Yaskawa INFORM job: aprem3TRJ3.JBI

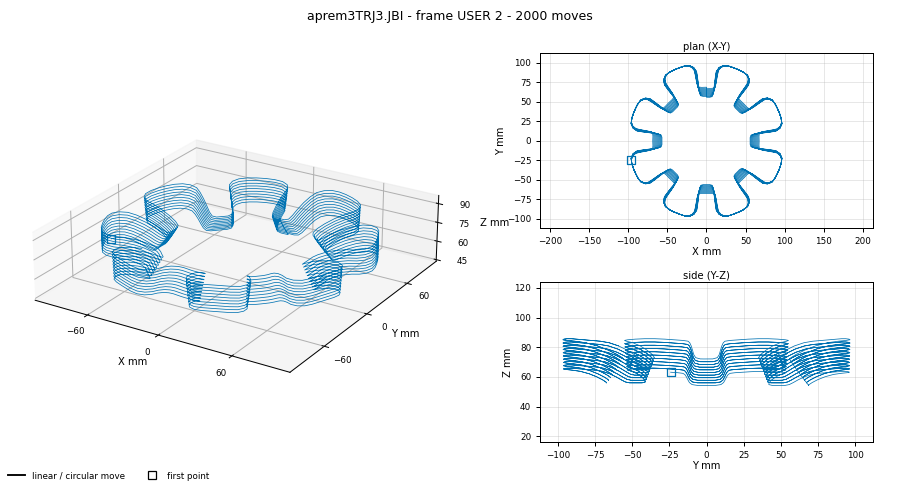
[picture p0: tool path of aprem3TRJ3.JBI in frame USER 2, 2000 of 2000 moves have a stored position in this frame; points joined in program order, loops and branches not executed]
/JOB
//NAME aprem3TRJ3
///FOLDERNAME DEMO
//POS
///NPOS 2000,0,2000,0,0,0
///USER 2
///TOOL 7
///POSTYPE USER
///RECTAN
///RCONF 1,0,0,0,0,0,0,0,0,0,0,0,0,0,0,0,0,0,0,0,0,0,0,0
C00000=-96.154,-24.159,63.210,179.7472,-2.4641,-10695.8962
C00001=-94.423,-19.246,62.877,177.2942,-4.1530,-10698.4794
C00002=-90.636,-15.942,62.469,172.7045,-3.4321,-10700.0243
C00003=-85.405,-14.621,61.698,172.2425,-1.7901,-10700.2854
C00004=-79.780,-13.569,60.151,174.0266,-1.3203,-10700.3475
C00005=-74.809,-12.586,58.158,176.9961,-0.7607,-10700.4499
C00006=-71.127,-11.507,56.252,-176.5790,1.2623,-10700.8103
C00007=-69.044,-9.699,54.888,-163.7838,26.3525,-10702.0037
C00008=-68.619,-6.200,54.350,-178.9508,38.3093,-10704.8371
C00009=-68.781,-2.945,54.326,177.7405,38.7530,-10707.5483
C00010=-68.843,0.000,54.342,179.9996,38.7765,-10710.0000
C00011=-68.781,2.945,54.326,-177.7401,38.7530,-10712.4517
C00012=-68.619,6.200,54.350,178.9482,38.3089,-10715.1629
C00013=-69.044,9.699,54.888,163.7840,26.3528,-10717.9963
C00014=-71.127,11.507,56.252,176.5790,1.2623,-10719.1897
C00015=-74.809,12.586,58.158,-176.9961,-0.7607,-10719.5501
C00016=-79.780,13.569,60.151,-174.0266,-1.3203,-10719.6525
C00017=-85.405,14.621,61.698,-172.2425,-1.7901,-10719.7146
C00018=-90.636,15.942,62.469,-172.7045,-3.4321,-10719.9757
C00019=-94.423,19.246,62.877,-177.2942,-4.1530,-10721.5206
C00020=-96.154,24.159,63.210,-179.7472,-2.4641,-10724.1038
C00021=-95.429,29.718,63.547,179.9546,-0.1514,-10727.2974
C00022=-93.512,35.416,63.770,179.9933,-0.0179,-10730.7433
C00023=-91.166,41.080,63.770,179.9921,-0.0174,-10734.2566
C00024=-88.493,46.465,63.547,179.9251,-0.1391,-10737.7026
C00025=-85.074,50.908,63.210,178.0786,-1.5643,-10740.8962
C00026=-80.376,53.158,62.877,175.1551,-1.0270,-10743.4793
C00027=-75.362,52.817,62.469,172.4279,2.7549,-10745.0245
C00028=-70.729,50.052,61.698,173.2462,4.2451,-10745.2855
C00029=-66.007,46.818,60.151,174.8410,3.3018,-10745.3476
C00030=-61.798,43.998,58.158,177.3380,1.5877,-10745.4495
C00031=-58.431,42.158,56.252,-176.6891,-1.5289,-10745.8105
C00032=-55.679,41.963,54.888,-150.9290,8.2296,-10747.0038
C00033=-52.905,44.137,54.350,-150.2488,28.6202,-10749.8372
C00034=-50.718,46.553,54.326,-151.6454,30.7727,-10752.5482
C00035=-48.679,48.679,54.342,-150.4014,29.5989,-10755.0000
C00036=-46.553,50.718,54.326,-149.2271,28.3544,-10757.4518
C00037=-44.137,52.905,54.350,-151.3816,29.7523,-10760.1628
C00038=-41.963,55.680,54.888,-171.7700,29.0711,-10762.9966
C00039=-42.158,58.431,56.252,178.4711,3.3109,-10764.1895
C00040=-43.998,61.798,58.158,-178.4123,-2.6620,-10764.5505
C00041=-46.818,66.007,60.151,-176.6982,-5.1590,-10764.6524
C00042=-50.052,70.729,61.698,-175.7549,-6.7538,-10764.7145
C00043=-52.817,75.362,62.469,-177.2451,-7.5721,-10764.9755
C00044=-53.158,80.376,62.877,178.9730,-4.8449,-10766.5207
C00045=-50.908,85.074,63.210,178.4357,-1.9214,-10769.1038
C00046=-46.465,88.493,63.547,179.8609,-0.0749,-10772.2974
C00047=-41.080,91.166,63.770,179.9826,-0.0079,-10775.7434
C00048=-35.416,93.512,63.770,179.9821,-0.0067,-10779.2567
C00049=-29.718,95.429,63.547,179.8486,-0.0454,-10782.7026
C00050=-24.159,96.154,63.210,177.5359,0.2528,-10785.8962
C00051=-19.246,94.423,62.877,175.8470,2.7058,-10788.4794
C00052=-15.942,90.636,62.469,176.5679,7.2955,-10790.0243
C00053=-14.621,85.405,61.698,178.2099,7.7575,-10790.2854
C00054=-13.569,79.780,60.151,178.6797,5.9734,-10790.3475
C00055=-12.586,74.809,58.158,179.2393,3.0039,-10790.4499
C00056=-11.507,71.127,56.252,-178.7377,-3.4210,-10790.8103
C00057=-9.699,69.044,54.888,-153.6472,-16.2160,-10792.0037
C00058=-6.200,68.619,54.350,-141.6911,-1.0518,-10794.8371
C00059=-2.945,68.781,54.326,-141.2470,2.2599,-10797.5483
C00060=0.000,68.843,54.342,-141.2235,-0.0004,-10800.0000
C00061=0.000,67.469,56.061,-141.5412,-0.0004,-10800.0000
C00062=2.820,67.413,56.044,-141.5636,-2.1988,-10802.3954
C00063=5.989,67.263,56.069,-142.0566,1.4090,-10805.0881
C00064=9.441,67.734,56.637,-154.9636,16.3668,-10807.9350
C00065=11.191,69.937,58.076,-179.1454,2.5065,-10809.0911
C00066=12.227,73.809,60.085,179.1943,-3.3815,-10809.4060
C00067=13.183,79.025,62.181,178.7261,-6.0865,-10809.4709
C00068=14.211,84.918,63.804,178.3204,-7.7435,-10809.5004
C00069=15.500,90.396,64.610,176.7328,-7.3164,-10809.7298
C00070=18.832,94.373,65.037,175.8897,-2.7823,-10811.2851
C00071=23.832,96.213,65.385,177.5484,-0.2740,-10813.9122
C00072=29.513,95.497,65.736,179.8479,0.0454,-10817.1736
C00073=35.347,93.539,65.969,179.9821,0.0067,-10820.7008
C00074=41.148,91.136,65.969,179.9826,0.0079,-10824.2992
C00075=46.658,88.395,65.736,179.8603,0.0754,-10827.8267
C00076=51.181,84.885,65.385,178.4595,1.9277,-10831.0877
C00077=53.416,80.048,65.037,179.0575,4.8686,-10833.7152
C00078=52.959,74.880,64.610,-177.1134,7.4719,-10835.2699
C00079=49.997,70.095,63.804,-175.6871,6.6669,-10835.4993
C00080=46.557,65.200,62.181,-176.5849,5.2066,-10835.5293
C00081=43.545,60.837,60.085,-178.1765,2.9610,-10835.5938
C00082=41.540,57.367,58.076,178.8310,-2.3765,-10835.9087
C00083=41.220,54.571,56.637,-173.0100,-28.2777,-10837.0654
C00084=43.327,51.796,56.069,-151.9006,-29.6278,-10839.9123
C00085=45.674,49.662,56.044,-149.5306,-28.1035,-10842.6047
C00086=47.708,47.708,56.061,-150.6800,-29.3196,-10845.0000
C00087=49.662,45.674,56.044,-151.8968,-30.4697,-10847.3953
C00088=51.797,43.327,56.069,-150.3712,-28.0975,-10850.0883
C00089=54.571,41.220,56.637,-151.7222,-6.9903,-10852.9346
C00090=57.367,41.540,58.076,-177.6235,1.1690,-10854.0913
C00091=60.837,43.545,60.085,177.0390,-1.8235,-10854.4062
C00092=65.200,46.557,62.181,174.7934,-3.4151,-10854.4707
C00093=70.095,49.997,63.804,173.3331,-4.3129,-10854.5007
C00094=74.880,52.959,64.610,172.5281,-2.8866,-10854.7301
C00095=80.048,53.416,65.037,175.1314,0.9425,-10856.2848
C00096=84.885,51.181,65.385,178.0723,1.5405,-10858.9123
C00097=88.395,46.658,65.736,179.9246,0.1397,-10862.1733
C00098=91.136,41.148,65.969,179.9921,0.0174,-10865.7008
C00099=93.539,35.347,65.969,179.9933,0.0179,-10869.2992
C00100=95.497,29.513,65.736,179.9546,0.1521,-10872.8264
C00101=96.213,23.832,65.385,-179.7260,2.4516,-10876.0878
C00102=94.373,18.832,65.037,-177.2177,4.1103,-10878.7149
C00103=90.396,15.500,64.610,-172.6836,3.2672,-10880.2702
C00104=84.918,14.211,63.804,-172.2565,1.6796,-10880.4996
C00105=79.025,13.183,62.181,-173.9135,1.2739,-10880.5291
C00106=73.809,12.227,60.085,-176.6185,0.8057,-10880.5940
C00107=69.937,11.191,58.076,177.4935,-0.8546,-10880.9089
C00108=67.734,9.441,56.637,163.6332,-25.0364,-10882.0650
C00109=67.263,5.989,56.069,178.5910,-37.9434,-10884.9119
C00110=67.413,2.820,56.044,-177.8012,-38.4364,-10887.6046
C00111=67.469,0.000,56.061,-179.9996,-38.4588,-10890.0000
C00112=67.413,-2.820,56.044,177.8008,-38.4364,-10892.3954
C00113=67.263,-5.989,56.069,-178.5883,-37.9429,-10895.0881
C00114=67.734,-9.441,56.637,-163.6333,-25.0366,-10897.9350
C00115=69.937,-11.191,58.076,-177.4935,-0.8546,-10899.0911
C00116=73.809,-12.227,60.085,176.6185,0.8057,-10899.4060
C00117=79.025,-13.183,62.181,173.9135,1.2739,-10899.4709
C00118=84.918,-14.211,63.804,172.2565,1.6796,-10899.5004
C00119=90.396,-15.500,64.610,172.6836,3.2672,-10899.7298
C00120=94.373,-18.832,65.037,177.2177,4.1103,-10901.2851
C00121=96.213,-23.832,65.385,179.7260,2.4516,-10903.9122
C00122=95.497,-29.513,65.736,-179.9546,0.1521,-10907.1736
C00123=93.539,-35.347,65.969,-179.9933,0.0179,-10910.7008
C00124=91.136,-41.148,65.969,-179.9921,0.0174,-10914.2992
C00125=88.395,-46.658,65.736,-179.9246,0.1397,-10917.8267
C00126=84.885,-51.181,65.385,-178.0723,1.5405,-10921.0877
C00127=80.048,-53.416,65.037,-175.1314,0.9425,-10923.7152
C00128=74.880,-52.959,64.610,-172.5281,-2.8866,-10925.2699
C00129=70.095,-49.997,63.804,-173.3331,-4.3129,-10925.4993
C00130=65.200,-46.557,62.181,-174.7934,-3.4151,-10925.5293
C00131=60.837,-43.545,60.085,-177.0390,-1.8235,-10925.5938
C00132=57.367,-41.540,58.076,177.6235,1.1690,-10925.9087
C00133=54.571,-41.220,56.637,151.7223,-6.9900,-10927.0654
C00134=51.796,-43.327,56.069,150.3722,-28.0994,-10929.9123
C00135=49.662,-45.674,56.044,151.8965,-30.4694,-10932.6047
C00136=47.708,-47.708,56.061,150.6804,-29.3200,-10935.0000
C00137=45.674,-49.662,56.044,149.5303,-28.1032,-10937.3953
C00138=43.327,-51.797,56.069,151.9025,-29.6288,-10940.0883
C00139=41.220,-54.571,56.637,173.0097,-28.2778,-10942.9346
C00140=41.540,-57.367,58.076,-178.8310,-2.3765,-10944.0913
C00141=43.545,-60.837,60.085,178.1765,2.9610,-10944.4062
C00142=46.557,-65.200,62.181,176.5849,5.2066,-10944.4707
C00143=49.997,-70.095,63.804,175.6871,6.6669,-10944.5007
C00144=52.959,-74.880,64.610,177.1134,7.4719,-10944.7301
C00145=53.416,-80.048,65.037,-179.0575,4.8686,-10946.2848
C00146=51.181,-84.885,65.385,-178.4595,1.9277,-10948.9123
C00147=46.658,-88.395,65.736,-179.8603,0.0754,-10952.1733
C00148=41.148,-91.136,65.969,-179.9826,0.0079,-10955.7008
C00149=35.347,-93.539,65.969,-179.9821,0.0067,-10959.2992
C00150=29.513,-95.497,65.736,-179.8479,0.0454,-10962.8264
C00151=23.832,-96.213,65.385,-177.5484,-0.2740,-10966.0878
C00152=18.832,-94.373,65.037,-175.8897,-2.7823,-10968.7149
C00153=15.500,-90.396,64.610,-176.7328,-7.3164,-10970.2702
C00154=14.211,-84.918,63.804,-178.3204,-7.7435,-10970.4996
C00155=13.183,-79.025,62.181,-178.7261,-6.0865,-10970.5291
C00156=12.227,-73.809,60.085,-179.1943,-3.3815,-10970.5940
C00157=11.191,-69.937,58.076,179.1454,2.5065,-10970.9089
C00158=9.441,-67.734,56.637,154.9636,16.3668,-10972.0650
C00159=5.989,-67.263,56.069,142.0566,1.4090,-10974.9119
C00160=2.820,-67.413,56.044,141.5636,-2.1988,-10977.6046
C00161=0.000,-67.469,56.061,141.5412,-0.0004,-10980.0000
C00162=0.000,-67.469,56.061,141.5412,-0.0004,-10980.0000
C00163=-2.820,-67.413,56.044,141.5636,2.1992,-10982.3954
C00164=-5.989,-67.263,56.069,142.0571,-1.4117,-10985.0881
C00165=-9.441,-67.734,56.637,154.9634,-16.3667,-10987.9350
C00166=-11.191,-69.937,58.076,179.1454,-2.5065,-10989.0911
C00167=-12.227,-73.809,60.085,-179.1943,3.3815,-10989.4060
C00168=-13.183,-79.025,62.181,-178.7261,6.0865,-10989.4709
C00169=-14.211,-84.918,63.804,-178.3204,7.7435,-10989.5004
C00170=-15.500,-90.396,64.610,-176.7328,7.3164,-10989.7298
C00171=-18.832,-94.373,65.037,-175.8897,2.7823,-10991.2851
C00172=-23.832,-96.213,65.385,-177.5484,0.2740,-10993.9122
C00173=-29.513,-95.497,65.736,-179.8479,-0.0454,-10997.1736
C00174=-35.347,-93.539,65.969,-179.9821,-0.0067,-11000.7008
C00175=-41.148,-91.136,65.969,-179.9826,-0.0079,-11004.2992
C00176=-46.658,-88.395,65.736,-179.8603,-0.0754,-11007.8267
C00177=-51.181,-84.885,65.385,-178.4595,-1.9277,-11011.0877
C00178=-53.416,-80.048,65.037,-179.0575,-4.8686,-11013.7152
C00179=-52.959,-74.880,64.610,177.1134,-7.4719,-11015.2699
C00180=-49.997,-70.095,63.804,175.6871,-6.6669,-11015.4993
C00181=-46.557,-65.200,62.181,176.5849,-5.2066,-11015.5293
C00182=-43.545,-60.837,60.085,178.1765,-2.9610,-11015.5938
C00183=-41.540,-57.367,58.076,-178.8310,2.3765,-11015.9087
C00184=-41.220,-54.571,56.637,173.0100,28.2777,-11017.0654
C00185=-43.327,-51.796,56.069,151.9006,29.6278,-11019.9123
C00186=-45.674,-49.662,56.044,149.5306,28.1035,-11022.6047
C00187=-47.708,-47.708,56.061,150.6800,29.3196,-11025.0000
C00188=-49.662,-45.674,56.044,151.8968,30.4697,-11027.3953
C00189=-51.797,-43.327,56.069,150.3712,28.0975,-11030.0883
C00190=-54.571,-41.220,56.637,151.7222,6.9903,-11032.9346
C00191=-57.367,-41.540,58.076,177.6235,-1.1690,-11034.0913
C00192=-60.837,-43.545,60.085,-177.0390,1.8235,-11034.4062
C00193=-65.200,-46.557,62.181,-174.7934,3.4151,-11034.4707
C00194=-70.095,-49.997,63.804,-173.3331,4.3129,-11034.5007
C00195=-74.880,-52.959,64.610,-172.5281,2.8866,-11034.7301
C00196=-80.048,-53.416,65.037,-175.1314,-0.9425,-11036.2848
C00197=-84.885,-51.181,65.385,-178.0723,-1.5405,-11038.9123
C00198=-88.395,-46.658,65.736,-179.9246,-0.1397,-11042.1733
C00199=-91.136,-41.148,65.969,-179.9921,-0.0174,-11045.7008
C00200=-93.539,-35.347,65.969,-179.9933,-0.0179,-11049.2992
C00201=-95.497,-29.513,65.736,-179.9546,-0.1521,-11052.8264
C00202=-96.213,-23.832,65.385,179.7260,-2.4516,-11056.0878
C00203=-94.373,-18.832,65.037,177.2177,-4.1103,-11058.7149
C00204=-90.396,-15.500,64.610,172.6836,-3.2672,-11060.2702
C00205=-84.918,-14.211,63.804,172.2565,-1.6796,-11060.4996
C00206=-79.025,-13.183,62.181,173.9135,-1.2739,-11060.5291
C00207=-73.809,-12.227,60.085,176.6185,-0.8057,-11060.5940
C00208=-69.937,-11.191,58.076,-177.4935,0.8546,-11060.9089
C00209=-67.734,-9.441,56.637,-163.6332,25.0364,-11062.0650
C00210=-67.263,-5.989,56.069,-178.5910,37.9434,-11064.9119
C00211=-67.413,-2.820,56.044,177.8012,38.4364,-11067.6046
C00212=-67.469,0.000,56.061,179.9996,38.4588,-11070.0000
C00213=-67.413,2.820,56.044,-177.8008,38.4364,-11072.3954
C00214=-67.263,5.989,56.069,178.5883,37.9429,-11075.0881
C00215=-67.734,9.441,56.637,163.6333,25.0366,-11077.9350
C00216=-69.937,11.191,58.076,177.4935,0.8546,-11079.0911
C00217=-73.809,12.227,60.085,-176.6185,-0.8057,-11079.4060
C00218=-79.025,13.183,62.181,-173.9135,-1.2739,-11079.4709
C00219=-84.918,14.211,63.804,-172.2565,-1.6796,-11079.5004
C00220=-90.396,15.500,64.610,-172.6836,-3.2672,-11079.7298
C00221=-94.373,18.832,65.037,-177.2177,-4.1103,-11081.2851
C00222=-96.213,23.832,65.385,-179.7260,-2.4516,-11083.9122
C00223=-95.497,29.513,65.736,179.9546,-0.1521,-11087.1736
C00224=-93.539,35.347,65.969,179.9933,-0.0179,-11090.7008
C00225=-91.136,41.148,65.969,179.9921,-0.0174,-11094.2992
C00226=-88.395,46.658,65.736,179.9246,-0.1397,-11097.8267
C00227=-84.885,51.181,65.385,178.0723,-1.5405,-11101.0877
C00228=-80.048,53.416,65.037,175.1314,-0.9425,-11103.7152
C00229=-74.880,52.959,64.610,172.5281,2.8866,-11105.2699
C00230=-70.095,49.997,63.804,173.3331,4.3129,-11105.4993
C00231=-65.200,46.557,62.181,174.7934,3.4151,-11105.5293
C00232=-60.837,43.545,60.085,177.0390,1.8235,-11105.5938
C00233=-57.367,41.540,58.076,-177.6235,-1.1690,-11105.9087
C00234=-54.571,41.220,56.637,-151.7223,6.9900,-11107.0654
C00235=-51.796,43.327,56.069,-150.3722,28.0994,-11109.9123
C00236=-49.662,45.674,56.044,-151.8965,30.4694,-11112.6047
C00237=-47.708,47.708,56.061,-150.6804,29.3200,-11115.0000
C00238=-45.674,49.662,56.044,-149.5303,28.1032,-11117.3953
C00239=-43.327,51.797,56.069,-151.9025,29.6288,-11120.0883
C00240=-41.220,54.571,56.637,-173.0097,28.2778,-11122.9346
C00241=-41.540,57.367,58.076,178.8310,2.3765,-11124.0913
C00242=-43.545,60.837,60.085,-178.1765,-2.9610,-11124.4062
C00243=-46.557,65.200,62.181,-176.5849,-5.2066,-11124.4707
C00244=-49.997,70.095,63.804,-175.6871,-6.6669,-11124.5007
C00245=-52.959,74.880,64.610,-177.1134,-7.4719,-11124.7301
C00246=-53.416,80.048,65.037,179.0575,-4.8686,-11126.2848
C00247=-51.181,84.885,65.385,178.4595,-1.9277,-11128.9123
C00248=-46.658,88.395,65.736,179.8603,-0.0754,-11132.1733
C00249=-41.148,91.136,65.969,179.9826,-0.0079,-11135.7008
C00250=-35.347,93.539,65.969,179.9821,-0.0067,-11139.2992
C00251=-29.513,95.497,65.736,179.8479,-0.0454,-11142.8264
C00252=-23.832,96.213,65.385,177.5484,0.2740,-11146.0878
C00253=-18.832,94.373,65.037,175.8897,2.7823,-11148.7149
C00254=-15.500,90.396,64.610,176.7328,7.3164,-11150.2702
C00255=-14.211,84.918,63.804,178.3204,7.7435,-11150.4996
C00256=-13.183,79.025,62.181,178.7261,6.0865,-11150.5291
C00257=-12.227,73.809,60.085,179.1943,3.3815,-11150.5940
C00258=-11.191,69.937,58.076,-179.1454,-2.5065,-11150.9089
C00259=-9.441,67.734,56.637,-154.9634,-16.3667,-11152.0650
C00260=-5.989,67.263,56.069,-142.0571,-1.4117,-11154.9119
C00261=-2.820,67.413,56.044,-141.5636,2.1992,-11157.6046
C00262=0.000,67.469,56.061,-141.5412,-0.0004,-11160.0000
C00263=0.000,66.107,57.788,-141.9405,-0.0005,-11160.0000
C00264=2.695,66.055,57.771,-141.9617,-2.1301,-11162.3363
C00265=5.779,65.917,57.797,-142.5088,1.7632,-11165.0104
C00266=9.185,66.436,58.394,-156.3340,16.3865,-11167.8714
C00267=10.880,68.762,59.909,-179.4729,1.6691,-11168.9912
C00268=11.874,72.826,62.021,179.1708,-3.6886,-11169.2604
C00269=12.805,78.288,64.219,178.7806,-6.1350,-11169.2892
C00270=13.814,84.445,65.915,178.4333,-7.6593,-11169.2905
C00271=15.073,90.163,66.756,176.9116,-7.2599,-11169.4907
C00272=18.432,94.325,67.200,175.9710,-2.8231,-11171.0568
C00273=23.517,96.271,67.561,177.5835,-0.2906,-11173.7273
C00274=29.315,95.562,67.927,179.8488,0.0450,-11177.0541
C00275=35.280,93.564,68.167,179.9823,0.0066,-11180.6599
C00276=41.213,91.107,68.167,179.9828,0.0078,-11184.3400
C00277=46.844,88.301,67.927,179.8613,0.0751,-11187.9461
C00278=51.445,84.703,67.561,178.4961,1.9145,-11191.2727
C00279=53.664,79.731,67.200,179.1443,4.8399,-11193.9430
C00280=53.097,74.413,66.756,-177.0274,7.3072,-11195.5096
C00281=49.944,69.479,65.915,-175.6680,6.5281,-11195.7099
C00282=46.303,64.413,64.219,-176.5119,5.2027,-11195.7103
C00283=43.100,59.892,62.021,-177.9754,3.1949,-11195.7399
C00284=40.929,56.315,59.909,179.1922,-1.5529,-11196.0092
C00285=40.483,53.472,58.394,-174.1779,-27.3765,-11197.1289
C00286=42.524,50.697,57.797,-152.4966,-29.4307,-11199.9895
C00287=44.802,48.614,57.771,-149.9071,-27.7853,-11202.6632
C00288=46.745,46.745,57.788,-151.0292,-28.9702,-11205.0000
C00289=48.613,44.802,57.771,-152.2149,-30.0932,-11207.3362
C00290=50.697,42.524,57.797,-150.5682,-27.5015,-11210.0105
C00291=53.472,40.483,58.395,-152.6235,-5.8223,-11212.8711
C00292=56.315,40.929,59.909,-178.4471,0.8078,-11213.9908
C00293=59.892,43.100,62.021,176.8051,-2.0246,-11214.2601
C00294=64.413,46.303,64.219,174.7973,-3.4881,-11214.2897
C00295=69.479,49.944,65.915,173.4719,-4.3320,-11214.2901
C00296=74.413,53.097,66.756,172.6928,-2.9726,-11214.4904
C00297=79.731,53.664,67.200,175.1601,0.8557,-11216.0570
C00298=84.703,51.445,67.561,178.0855,1.5039,-11218.7273
C00299=88.301,46.844,67.927,179.9249,0.1387,-11222.0539
C00300=91.107,41.213,68.167,179.9922,0.0172,-11225.6600
C00301=93.564,35.280,68.167,179.9934,0.0177,-11229.3401
C00302=95.562,29.315,67.927,179.9550,0.1512,-11232.9459
C00303=96.271,23.517,67.561,-179.7094,2.4165,-11236.2727
C00304=94.325,18.432,67.200,-177.1769,4.0290,-11238.9432
C00305=90.163,15.073,66.756,-172.7401,3.0884,-11240.5093
C00306=84.445,13.814,65.915,-172.3407,1.5667,-11240.7095
C00307=78.288,12.805,64.219,-173.8650,1.2194,-11240.7108
C00308=72.826,11.874,62.021,-176.3114,0.8292,-11240.7396
C00309=68.762,10.880,59.909,178.3309,-0.5271,-11241.0088
C00310=66.436,9.185,58.394,163.6135,-23.6660,-11242.1286
C00311=65.917,5.779,57.797,178.2368,-37.4912,-11244.9896
C00312=66.055,2.695,57.771,-177.8699,-38.0383,-11247.6637
C00313=66.107,0.000,57.788,-179.9995,-38.0595,-11250.0000
C00314=66.055,-2.695,57.771,177.8693,-38.0383,-11252.3363
C00315=65.917,-5.780,57.797,-178.2340,-37.4907,-11255.0112
C00316=66.436,-9.185,58.395,-163.6136,-23.6662,-11257.8714
C00317=68.762,-10.880,59.909,-178.3309,-0.5271,-11258.9912
C00318=72.826,-11.874,62.021,176.3114,0.8292,-11259.2604
C00319=78.288,-12.805,64.219,173.8650,1.2194,-11259.2892
C00320=84.445,-13.814,65.915,172.3407,1.5667,-11259.2905
C00321=90.163,-15.073,66.756,172.7401,3.0884,-11259.4907
C00322=94.325,-18.432,67.200,177.1769,4.0290,-11261.0568
C00323=96.271,-23.517,67.561,179.7094,2.4165,-11263.7273
C00324=95.562,-29.315,67.927,-179.9550,0.1512,-11267.0541
C00325=93.564,-35.280,68.167,-179.9934,0.0177,-11270.6599
C00326=91.107,-41.213,68.167,-179.9922,0.0172,-11274.3400
C00327=88.301,-46.844,67.927,-179.9249,0.1387,-11277.9461
C00328=84.703,-51.445,67.561,-178.0855,1.5039,-11281.2727
C00329=79.731,-53.664,67.200,-175.1601,0.8557,-11283.9430
C00330=74.413,-53.097,66.756,-172.6928,-2.9726,-11285.5096
C00331=69.479,-49.944,65.915,-173.4719,-4.3320,-11285.7099
C00332=64.413,-46.303,64.219,-174.7973,-3.4881,-11285.7103
C00333=59.892,-43.100,62.021,-176.8051,-2.0246,-11285.7399
C00334=56.315,-40.929,59.909,178.4471,0.8078,-11286.0092
C00335=53.472,-40.483,58.394,152.6235,-5.8221,-11287.1289
C00336=50.697,-42.524,57.797,150.5693,-27.5034,-11289.9895
C00337=48.614,-44.802,57.771,152.2147,-30.0929,-11292.6632
C00338=46.745,-46.745,57.788,151.0298,-28.9708,-11295.0000
C00339=44.802,-48.613,57.771,149.9068,-27.7851,-11297.3362
C00340=42.524,-50.697,57.797,152.4985,-29.4318,-11300.0105
C00341=40.483,-53.472,58.395,174.1777,-27.3765,-11302.8711
C00342=40.929,-56.315,59.909,-179.1922,-1.5529,-11303.9908
C00343=43.100,-59.892,62.021,177.9754,3.1949,-11304.2601
C00344=46.303,-64.413,64.219,176.5119,5.2027,-11304.2897
C00345=49.944,-69.479,65.915,175.6680,6.5281,-11304.2901
C00346=53.097,-74.413,66.756,177.0274,7.3072,-11304.4904
C00347=53.664,-79.731,67.200,-179.1443,4.8399,-11306.0570
C00348=51.445,-84.703,67.561,-178.4961,1.9145,-11308.7273
C00349=46.844,-88.301,67.927,-179.8613,0.0751,-11312.0539
C00350=41.213,-91.107,68.167,-179.9828,0.0078,-11315.6600
C00351=35.280,-93.564,68.167,-179.9823,0.0066,-11319.3401
C00352=29.315,-95.562,67.927,-179.8488,0.0450,-11322.9459
C00353=23.517,-96.271,67.561,-177.5835,-0.2906,-11326.2727
C00354=18.432,-94.325,67.200,-175.9710,-2.8231,-11328.9432
C00355=15.073,-90.163,66.756,-176.9116,-7.2599,-11330.5093
C00356=13.814,-84.445,65.915,-178.4333,-7.6593,-11330.7095
C00357=12.805,-78.288,64.219,-178.7806,-6.1350,-11330.7108
C00358=11.874,-72.826,62.021,-179.1708,-3.6886,-11330.7396
C00359=10.880,-68.762,59.909,179.4729,1.6691,-11331.0088
C00360=9.185,-66.436,58.394,156.3340,16.3865,-11332.1286
C00361=5.779,-65.917,57.797,142.5088,1.7632,-11334.9896
C00362=2.695,-66.055,57.771,141.9617,-2.1301,-11337.6637
C00363=0.000,-66.107,57.788,141.9405,-0.0005,-11340.0000
C00364=0.000,-66.107,57.788,141.9405,-0.0005,-11340.0000
C00365=-2.695,-66.055,57.771,141.9617,2.1307,-11342.3363
C00366=-5.780,-65.917,57.797,142.5093,-1.7660,-11345.0112
C00367=-9.185,-66.436,58.395,156.3338,-16.3864,-11347.8714
C00368=-10.880,-68.762,59.909,179.4729,-1.6691,-11348.9912
C00369=-11.874,-72.826,62.021,-179.1708,3.6886,-11349.2604
C00370=-12.805,-78.288,64.219,-178.7806,6.1350,-11349.2892
C00371=-13.814,-84.445,65.915,-178.4333,7.6593,-11349.2905
C00372=-15.073,-90.163,66.756,-176.9116,7.2599,-11349.4907
C00373=-18.432,-94.325,67.200,-175.9710,2.8231,-11351.0568
C00374=-23.517,-96.271,67.561,-177.5835,0.2906,-11353.7273
C00375=-29.315,-95.562,67.927,-179.8488,-0.0450,-11357.0541
C00376=-35.280,-93.564,68.167,-179.9823,-0.0066,-11360.6599
C00377=-41.213,-91.107,68.167,-179.9828,-0.0078,-11364.3400
C00378=-46.844,-88.301,67.927,-179.8613,-0.0751,-11367.9461
C00379=-51.445,-84.703,67.561,-178.4961,-1.9145,-11371.2727
C00380=-53.664,-79.731,67.200,-179.1443,-4.8399,-11373.9430
C00381=-53.097,-74.413,66.756,177.0274,-7.3072,-11375.5096
C00382=-49.944,-69.479,65.915,175.6680,-6.5281,-11375.7099
C00383=-46.303,-64.413,64.219,176.5119,-5.2027,-11375.7103
C00384=-43.100,-59.892,62.021,177.9754,-3.1949,-11375.7399
C00385=-40.929,-56.315,59.909,-179.1922,1.5529,-11376.0092
C00386=-40.483,-53.472,58.394,174.1779,27.3765,-11377.1289
C00387=-42.524,-50.697,57.797,152.4966,29.4307,-11379.9895
C00388=-44.802,-48.614,57.771,149.9071,27.7853,-11382.6632
C00389=-46.745,-46.745,57.788,151.0292,28.9702,-11385.0000
C00390=-48.613,-44.802,57.771,152.2149,30.0932,-11387.3362
C00391=-50.697,-42.524,57.797,150.5682,27.5015,-11390.0105
C00392=-53.472,-40.483,58.395,152.6235,5.8223,-11392.8711
C00393=-56.315,-40.929,59.909,178.4471,-0.8078,-11393.9908
C00394=-59.892,-43.100,62.021,-176.8051,2.0246,-11394.2601
C00395=-64.413,-46.303,64.219,-174.7973,3.4881,-11394.2897
C00396=-69.479,-49.944,65.915,-173.4719,4.3320,-11394.2901
C00397=-74.413,-53.097,66.756,-172.6928,2.9726,-11394.4904
C00398=-79.731,-53.664,67.200,-175.1601,-0.8557,-11396.0570
C00399=-84.703,-51.445,67.561,-178.0855,-1.5039,-11398.7273
C00400=-88.301,-46.844,67.927,-179.9249,-0.1387,-11402.0539
C00401=-91.107,-41.213,68.167,-179.9922,-0.0172,-11405.6600
C00402=-93.564,-35.280,68.167,-179.9934,-0.0177,-11409.3401
C00403=-95.562,-29.315,67.927,-179.9550,-0.1512,-11412.9459
C00404=-96.271,-23.517,67.561,179.7094,-2.4165,-11416.2727
C00405=-94.325,-18.432,67.200,177.1769,-4.0290,-11418.9432
C00406=-90.163,-15.073,66.756,172.7401,-3.0884,-11420.5093
C00407=-84.445,-13.814,65.915,172.3407,-1.5667,-11420.7095
C00408=-78.288,-12.805,64.219,173.8650,-1.2194,-11420.7108
C00409=-72.826,-11.874,62.021,176.3114,-0.8292,-11420.7396
C00410=-68.762,-10.880,59.909,-178.3309,0.5271,-11421.0088
C00411=-66.436,-9.185,58.394,-163.6135,23.6660,-11422.1286
C00412=-65.917,-5.779,57.797,-178.2368,37.4912,-11424.9896
C00413=-66.055,-2.695,57.771,177.8699,38.0383,-11427.6637
C00414=-66.107,0.000,57.788,179.9995,38.0595,-11430.0000
C00415=-66.055,2.695,57.771,-177.8693,38.0383,-11432.3363
C00416=-65.917,5.780,57.797,178.2340,37.4907,-11435.0112
C00417=-66.436,9.185,58.395,163.6136,23.6662,-11437.8714
C00418=-68.762,10.880,59.909,178.3309,0.5271,-11438.9912
C00419=-72.826,11.874,62.021,-176.3114,-0.8292,-11439.2604
C00420=-78.288,12.805,64.219,-173.8650,-1.2194,-11439.2892
C00421=-84.445,13.814,65.915,-172.3407,-1.5667,-11439.2905
C00422=-90.163,15.073,66.756,-172.7401,-3.0884,-11439.4907
C00423=-94.325,18.432,67.200,-177.1769,-4.0290,-11441.0568
C00424=-96.271,23.517,67.561,-179.7094,-2.4165,-11443.7273
C00425=-95.562,29.315,67.927,179.9550,-0.1512,-11447.0541
C00426=-93.564,35.280,68.167,179.9934,-0.0177,-11450.6599
C00427=-91.107,41.213,68.167,179.9922,-0.0172,-11454.3400
C00428=-88.301,46.844,67.927,179.9249,-0.1387,-11457.9461
C00429=-84.703,51.445,67.561,178.0855,-1.5039,-11461.2727
C00430=-79.731,53.664,67.200,175.1601,-0.8557,-11463.9430
C00431=-74.413,53.097,66.756,172.6928,2.9726,-11465.5096
C00432=-69.479,49.944,65.915,173.4719,4.3320,-11465.7099
C00433=-64.413,46.303,64.219,174.7973,3.4881,-11465.7103
C00434=-59.892,43.100,62.021,176.8051,2.0246,-11465.7399
C00435=-56.315,40.929,59.909,-178.4471,-0.8078,-11466.0092
C00436=-53.472,40.483,58.394,-152.6235,5.8221,-11467.1289
C00437=-50.697,42.524,57.797,-150.5693,27.5034,-11469.9895
C00438=-48.614,44.802,57.771,-152.2147,30.0929,-11472.6632
C00439=-46.745,46.745,57.788,-151.0298,28.9708,-11475.0000
C00440=-44.802,48.613,57.771,-149.9068,27.7851,-11477.3362
C00441=-42.524,50.697,57.797,-152.4985,29.4318,-11480.0105
C00442=-40.483,53.472,58.395,-174.1777,27.3765,-11482.8711
C00443=-40.929,56.315,59.909,179.1922,1.5529,-11483.9908
C00444=-43.100,59.892,62.021,-177.9754,-3.1949,-11484.2601
C00445=-46.303,64.413,64.219,-176.5119,-5.2027,-11484.2897
C00446=-49.944,69.479,65.915,-175.6680,-6.5281,-11484.2901
C00447=-53.097,74.413,66.756,-177.0274,-7.3072,-11484.4904
C00448=-53.664,79.731,67.200,179.1443,-4.8399,-11486.0570
C00449=-51.445,84.703,67.561,178.4961,-1.9145,-11488.7273
C00450=-46.844,88.301,67.927,179.8613,-0.0751,-11492.0539
C00451=-41.213,91.107,68.167,179.9828,-0.0078,-11495.6600
C00452=-35.280,93.564,68.167,179.9823,-0.0066,-11499.3401
C00453=-29.315,95.562,67.927,179.8488,-0.0450,-11502.9459
C00454=-23.517,96.271,67.561,177.5835,0.2906,-11506.2727
C00455=-18.432,94.325,67.200,175.9710,2.8231,-11508.9432
C00456=-15.073,90.163,66.756,176.9116,7.2599,-11510.5093
C00457=-13.814,84.445,65.915,178.4333,7.6593,-11510.7095
C00458=-12.805,78.288,64.219,178.7806,6.1350,-11510.7108
C00459=-11.874,72.826,62.021,179.1708,3.6886,-11510.7396
C00460=-10.880,68.762,59.909,-179.4729,-1.6691,-11511.0088
C00461=-9.185,66.436,58.395,-156.3338,-16.3864,-11512.1286
C00462=-5.780,65.917,57.797,-142.5093,-1.7660,-11514.9888
C00463=-2.695,66.055,57.771,-141.9617,2.1307,-11517.6637
C00464=0.000,66.107,57.788,-141.9405,-0.0005,-11520.0000
C00465=0.000,64.758,59.526,-142.4254,-0.0006,-11520.0000
C00466=2.572,64.710,59.508,-142.4454,-2.0536,-11522.2761
C00467=5.572,64.584,59.535,-143.0512,2.1076,-11524.9310
C00468=8.932,65.152,60.163,-157.7440,16.2795,-11527.8063
C00469=10.572,67.603,61.754,-179.7324,0.9128,-11528.8881
C00470=11.527,71.864,63.969,179.1649,-3.9269,-11529.1126
C00471=12.439,77.571,66.266,178.8415,-6.1204,-11529.1102
C00472=13.430,83.988,68.033,178.5474,-7.5065,-11529.0849
C00473=14.662,89.940,68.906,177.1014,-7.1283,-11529.2589
C00474=18.048,94.279,69.366,176.0893,-2.8270,-11530.8371
C00475=23.215,96.325,69.740,177.6414,-0.3022,-11533.5503
C00476=29.126,95.625,70.117,179.8514,0.0441,-11536.9400
C00477=35.216,93.589,70.366,179.9827,0.0065,-11540.6205
C00478=41.276,91.079,70.366,179.9832,0.0077,-11544.3795
C00479=47.022,88.212,70.117,179.8638,0.0739,-11548.0601
C00480=51.697,84.528,69.740,178.5453,1.8817,-11551.4498
C00481=53.903,79.427,69.366,179.2311,4.7592,-11554.1627
C00482=53.229,73.964,68.906,-176.9875,7.0817,-11555.7411
C00483=49.892,68.885,68.033,-175.6970,6.3398,-11555.9150
C00484=46.056,63.647,66.266,-176.4794,5.1497,-11555.8901
C00485=42.664,58.966,63.969,-177.8105,3.3678,-11555.8871
C00486=40.327,55.279,61.754,179.5437,-0.8347,-11556.1114
C00487=39.754,52.385,60.163,-175.2625,-26.3754,-11557.1942
C00488=41.728,49.608,59.535,-153.1683,-29.1561,-11560.0690
C00489=43.938,47.576,59.508,-150.3598,-27.3976,-11562.7235
C00490=45.791,45.791,59.526,-151.4514,-28.5479,-11565.0000
C00491=47.575,43.938,59.508,-152.6027,-29.6406,-11567.2759
C00492=49.608,41.728,59.535,-150.8429,-26.8297,-11569.9310
C00493=52.385,39.754,60.163,-153.6246,-4.7376,-11572.8058
C00494=55.279,40.327,61.754,-179.1653,0.4563,-11573.8886
C00495=58.966,42.664,63.969,176.6322,-2.1895,-11574.1129
C00496=63.647,46.056,66.266,174.8503,-3.5206,-11574.1099
C00497=68.885,49.892,68.033,173.6602,-4.3030,-11574.0850
C00498=73.964,53.229,68.906,172.9183,-3.0125,-11574.2589
C00499=79.427,53.903,69.366,175.2408,0.7689,-11575.8373
C00500=84.528,51.697,69.740,178.1183,1.4547,-11578.5502
C00501=88.212,47.022,70.117,179.9261,0.1362,-11581.9399
C00502=91.079,41.276,70.366,179.9923,0.0168,-11585.6205
C00503=93.589,35.216,70.366,179.9935,0.0173,-11589.3795
C00504=95.625,29.126,70.117,179.9559,0.1486,-11593.0600
C00505=96.325,23.215,69.740,-179.6978,2.3586,-11596.4497
C00506=94.279,18.048,69.366,-177.1730,3.9107,-11599.1629
C00507=89.940,14.662,68.906,-172.8717,2.8986,-11600.7411
C00508=83.988,13.430,68.033,-172.4935,1.4526,-11600.9151
C00509=77.571,12.439,66.266,-173.8796,1.1585,-11600.8898
C00510=71.864,11.527,63.969,-176.0731,0.8351,-11600.8874
C00511=67.603,10.572,61.754,179.0872,-0.2676,-11601.1119
C00512=65.152,8.932,60.163,163.7205,-22.2560,-11602.1937
C00513=64.584,5.572,59.535,177.8924,-36.9488,-11605.0690
C00514=64.710,2.572,59.508,-177.9464,-37.5546,-11607.7239
C00515=64.758,0.000,59.526,-179.9994,-37.5746,-11610.0000
C00516=64.710,-2.572,59.508,177.9458,-37.5546,-11612.2761
C00517=64.584,-5.572,59.535,-177.8896,-36.9483,-11614.9310
C00518=65.152,-8.932,60.163,-163.7206,-22.2560,-11617.8063
C00519=67.603,-10.572,61.754,-179.0872,-0.2676,-11618.8881
C00520=71.864,-11.527,63.969,176.0731,0.8351,-11619.1126
C00521=77.571,-12.439,66.266,173.8796,1.1585,-11619.1102
C00522=83.988,-13.430,68.033,172.4935,1.4526,-11619.0849
C00523=89.940,-14.662,68.906,172.8717,2.8986,-11619.2589
C00524=94.279,-18.048,69.366,177.1730,3.9107,-11620.8371
C00525=96.325,-23.215,69.740,179.6978,2.3586,-11623.5503
C00526=95.625,-29.126,70.117,-179.9559,0.1486,-11626.9400
C00527=93.589,-35.216,70.366,-179.9935,0.0173,-11630.6205
C00528=91.079,-41.276,70.366,-179.9923,0.0168,-11634.3795
C00529=88.212,-47.022,70.117,-179.9261,0.1362,-11638.0601
C00530=84.528,-51.697,69.740,-178.1183,1.4547,-11641.4498
C00531=79.427,-53.903,69.366,-175.2408,0.7689,-11644.1627
C00532=73.964,-53.229,68.906,-172.9183,-3.0125,-11645.7411
C00533=68.885,-49.892,68.033,-173.6602,-4.3030,-11645.9150
C00534=63.647,-46.056,66.266,-174.8503,-3.5206,-11645.8901
C00535=58.966,-42.664,63.969,-176.6322,-2.1895,-11645.8871
C00536=55.279,-40.327,61.754,179.1653,0.4563,-11646.1114
C00537=52.385,-39.754,60.163,153.6246,-4.7375,-11647.1942
C00538=49.608,-41.728,59.535,150.8439,-26.8317,-11650.0690
C00539=47.576,-43.938,59.508,152.6024,-29.6402,-11652.7235
C00540=45.791,-45.791,59.526,151.4521,-28.5486,-11655.0000
C00541=43.938,-47.575,59.508,150.3594,-27.3973,-11657.2759
C00542=41.728,-49.608,59.535,153.1703,-29.1571,-11659.9310
C00543=39.754,-52.385,60.163,175.2624,-26.3754,-11662.8058
C00544=40.327,-55.279,61.754,-179.5437,-0.8347,-11663.8886
C00545=42.664,-58.966,63.969,177.8105,3.3678,-11664.1129
C00546=46.056,-63.647,66.266,176.4794,5.1497,-11664.1099
C00547=49.892,-68.885,68.033,175.6970,6.3398,-11664.0850
C00548=53.229,-73.964,68.906,176.9875,7.0817,-11664.2589
C00549=53.903,-79.427,69.366,-179.2311,4.7592,-11665.8373
C00550=51.697,-84.528,69.740,-178.5453,1.8817,-11668.5502
C00551=47.022,-88.212,70.117,-179.8638,0.0739,-11671.9399
C00552=41.276,-91.079,70.366,-179.9832,0.0077,-11675.6205
C00553=35.216,-93.589,70.366,-179.9827,0.0065,-11679.3795
C00554=29.126,-95.625,70.117,-179.8514,0.0441,-11683.0600
C00555=23.215,-96.325,69.740,-177.6414,-0.3022,-11686.4497
C00556=18.048,-94.279,69.366,-176.0893,-2.8270,-11689.1629
C00557=14.662,-89.940,68.906,-177.1014,-7.1283,-11690.7411
C00558=13.430,-83.988,68.033,-178.5474,-7.5065,-11690.9151
C00559=12.439,-77.571,66.266,-178.8415,-6.1204,-11690.8898
C00560=11.527,-71.864,63.969,-179.1649,-3.9269,-11690.8874
C00561=10.572,-67.603,61.754,179.7324,0.9128,-11691.1119
C00562=8.932,-65.152,60.163,157.7440,16.2795,-11692.1937
C00563=5.572,-64.584,59.535,143.0512,2.1076,-11695.0690
C00564=2.572,-64.710,59.508,142.4454,-2.0536,-11697.7239
C00565=0.000,-64.758,59.526,142.4254,-0.0006,-11700.0000
C00566=0.000,-64.758,59.526,142.4254,-0.0006,-11700.0000
C00567=-2.572,-64.710,59.508,142.4454,2.0542,-11702.2761
C00568=-5.572,-64.584,59.535,143.0517,-2.1104,-11704.9310
C00569=-8.932,-65.152,60.163,157.7440,-16.2794,-11707.8063
C00570=-10.572,-67.603,61.754,179.7324,-0.9128,-11708.8881
C00571=-11.527,-71.864,63.969,-179.1649,3.9269,-11709.1126
C00572=-12.439,-77.571,66.266,-178.8415,6.1204,-11709.1102
C00573=-13.430,-83.988,68.033,-178.5474,7.5065,-11709.0849
C00574=-14.662,-89.940,68.906,-177.1014,7.1283,-11709.2589
C00575=-18.048,-94.279,69.366,-176.0893,2.8270,-11710.8371
C00576=-23.215,-96.325,69.740,-177.6414,0.3022,-11713.5503
C00577=-29.126,-95.625,70.117,-179.8514,-0.0441,-11716.9400
C00578=-35.216,-93.589,70.366,-179.9827,-0.0065,-11720.6205
C00579=-41.276,-91.079,70.366,-179.9832,-0.0077,-11724.3795
C00580=-47.022,-88.212,70.117,-179.8638,-0.0739,-11728.0601
C00581=-51.697,-84.528,69.740,-178.5453,-1.8817,-11731.4498
C00582=-53.903,-79.427,69.366,-179.2311,-4.7592,-11734.1627
C00583=-53.229,-73.964,68.906,176.9875,-7.0817,-11735.7411
C00584=-49.892,-68.885,68.033,175.6970,-6.3398,-11735.9150
C00585=-46.056,-63.647,66.266,176.4794,-5.1497,-11735.8901
C00586=-42.664,-58.966,63.969,177.8105,-3.3678,-11735.8871
C00587=-40.327,-55.279,61.754,-179.5437,0.8347,-11736.1114
C00588=-39.754,-52.385,60.163,175.2625,26.3754,-11737.1942
C00589=-41.728,-49.608,59.535,153.1683,29.1561,-11740.0690
C00590=-43.938,-47.576,59.508,150.3598,27.3976,-11742.7235
C00591=-45.791,-45.791,59.526,151.4514,28.5479,-11745.0000
C00592=-47.575,-43.938,59.508,152.6027,29.6406,-11747.2759
C00593=-49.608,-41.728,59.535,150.8429,26.8297,-11749.9310
C00594=-52.385,-39.754,60.163,153.6246,4.7376,-11752.8058
C00595=-55.279,-40.327,61.754,179.1653,-0.4563,-11753.8886
C00596=-58.966,-42.664,63.969,-176.6322,2.1895,-11754.1129
C00597=-63.647,-46.056,66.266,-174.8503,3.5206,-11754.1099
C00598=-68.885,-49.892,68.033,-173.6602,4.3030,-11754.0850
C00599=-73.964,-53.229,68.906,-172.9183,3.0125,-11754.2589
C00600=-79.427,-53.903,69.366,-175.2408,-0.7689,-11755.8373
C00601=-84.528,-51.697,69.740,-178.1183,-1.4547,-11758.5502
C00602=-88.212,-47.022,70.117,-179.9261,-0.1362,-11761.9399
C00603=-91.079,-41.276,70.366,-179.9923,-0.0168,-11765.6205
C00604=-93.589,-35.216,70.366,-179.9935,-0.0173,-11769.3795
C00605=-95.625,-29.126,70.117,-179.9559,-0.1486,-11773.0600
C00606=-96.325,-23.215,69.740,179.6978,-2.3586,-11776.4497
C00607=-94.279,-18.048,69.366,177.1730,-3.9107,-11779.1629
C00608=-89.940,-14.662,68.906,172.8717,-2.8986,-11780.7411
C00609=-83.988,-13.430,68.033,172.4935,-1.4526,-11780.9151
C00610=-77.571,-12.439,66.266,173.8796,-1.1585,-11780.8898
C00611=-71.864,-11.527,63.969,176.0731,-0.8351,-11780.8874
C00612=-67.603,-10.572,61.754,-179.0872,0.2676,-11781.1119
C00613=-65.152,-8.932,60.163,-163.7205,22.2560,-11782.1937
C00614=-64.584,-5.572,59.535,-177.8924,36.9488,-11785.0690
C00615=-64.710,-2.572,59.508,177.9464,37.5546,-11787.7239
C00616=-64.758,0.000,59.526,179.9994,37.5746,-11790.0000
C00617=-64.710,2.572,59.508,-177.9458,37.5546,-11792.2761
C00618=-64.584,5.572,59.535,177.8896,36.9483,-11794.9310
C00619=-65.152,8.932,60.163,163.7206,22.2560,-11797.8063
C00620=-67.603,10.572,61.754,179.0872,0.2676,-11798.8881
C00621=-71.864,11.527,63.969,-176.0731,-0.8351,-11799.1126
C00622=-77.571,12.439,66.266,-173.8796,-1.1585,-11799.1102
C00623=-83.988,13.430,68.033,-172.4935,-1.4526,-11799.0849
C00624=-89.940,14.662,68.906,-172.8717,-2.8986,-11799.2589
C00625=-94.279,18.048,69.366,-177.1730,-3.9107,-11800.8371
C00626=-96.325,23.215,69.740,-179.6978,-2.3586,-11803.5503
C00627=-95.625,29.126,70.117,179.9559,-0.1486,-11806.9400
C00628=-93.589,35.216,70.366,179.9935,-0.0173,-11810.6205
C00629=-91.079,41.276,70.366,179.9923,-0.0168,-11814.3795
C00630=-88.212,47.022,70.117,179.9261,-0.1362,-11818.0601
C00631=-84.528,51.697,69.740,178.1183,-1.4547,-11821.4498
C00632=-79.427,53.903,69.366,175.2408,-0.7689,-11824.1627
C00633=-73.964,53.229,68.906,172.9183,3.0125,-11825.7411
C00634=-68.885,49.892,68.033,173.6602,4.3030,-11825.9150
C00635=-63.647,46.056,66.266,174.8503,3.5206,-11825.8901
C00636=-58.966,42.664,63.969,176.6322,2.1895,-11825.8871
C00637=-55.279,40.327,61.754,-179.1653,-0.4563,-11826.1114
C00638=-52.385,39.754,60.163,-153.6246,4.7375,-11827.1942
C00639=-49.608,41.728,59.535,-150.8439,26.8317,-11830.0690
C00640=-47.576,43.938,59.508,-152.6024,29.6402,-11832.7235
C00641=-45.791,45.791,59.526,-151.4521,28.5486,-11835.0000
C00642=-43.938,47.575,59.508,-150.3594,27.3973,-11837.2759
C00643=-41.728,49.608,59.535,-153.1703,29.1571,-11839.9310
C00644=-39.754,52.385,60.163,-175.2624,26.3754,-11842.8058
C00645=-40.327,55.279,61.754,179.5437,0.8347,-11843.8886
C00646=-42.664,58.966,63.969,-177.8105,-3.3678,-11844.1129
C00647=-46.056,63.647,66.266,-176.4794,-5.1497,-11844.1099
C00648=-49.892,68.885,68.033,-175.6970,-6.3398,-11844.0850
C00649=-53.229,73.964,68.906,-176.9875,-7.0817,-11844.2589
C00650=-53.903,79.427,69.366,179.2311,-4.7592,-11845.8373
C00651=-51.697,84.528,69.740,178.5453,-1.8817,-11848.5502
C00652=-47.022,88.212,70.117,179.8638,-0.0739,-11851.9399
C00653=-41.276,91.079,70.366,179.9832,-0.0077,-11855.6205
C00654=-35.216,93.589,70.366,179.9827,-0.0065,-11859.3795
C00655=-29.126,95.625,70.117,179.8514,-0.0441,-11863.0600
C00656=-23.215,96.325,69.740,177.6414,0.3022,-11866.4497
C00657=-18.048,94.279,69.366,176.0893,2.8270,-11869.1629
C00658=-14.662,89.940,68.906,177.1014,7.1283,-11870.7411
C00659=-13.430,83.988,68.033,178.5474,7.5065,-11870.9151
C00660=-12.439,77.571,66.266,178.8415,6.1204,-11870.8898
C00661=-11.527,71.864,63.969,179.1649,3.9269,-11870.8874
C00662=-10.572,67.603,61.754,-179.7324,-0.9128,-11871.1119
C00663=-8.932,65.152,60.163,-157.7440,-16.2794,-11872.1937
C00664=-5.572,64.584,59.535,-143.0517,-2.1104,-11875.0690
C00665=-2.572,64.710,59.508,-142.4454,2.0542,-11877.7239
C00666=0.000,64.758,59.526,-142.4254,-0.0006,-11880.0000
C00667=0.000,63.425,61.276,-143.0012,-0.0007,-11880.0000
C00668=2.450,63.381,61.257,-143.0199,-1.9693,-11882.2137
C00669=5.367,63.268,61.285,-143.6888,2.4374,-11884.8488
C00670=8.682,63.886,61.945,-159.1792,16.0512,-11887.7390
C00671=10.270,66.465,63.612,-179.9346,0.2399,-11888.7837
C00672=11.189,70.924,65.929,179.1735,-4.0983,-11888.9651
C00673=12.084,76.878,68.324,178.9074,-6.0442,-11888.9329
C00674=13.063,83.550,70.157,178.6617,-7.2870,-11888.8862
C00675=14.270,89.726,71.060,177.3000,-6.9235,-11889.0366
C00676=17.683,94.235,71.535,176.2430,-2.7934,-11890.6278
C00677=22.929,96.378,71.920,177.7221,-0.3083,-11893.3823
C00678=28.946,95.684,72.309,179.8557,0.0426,-11896.8314
C00679=35.156,93.612,72.565,179.9833,0.0062,-11900.5837
C00680=41.335,91.053,72.565,179.9837,0.0074,-11904.4165
C00681=47.191,88.127,72.309,179.8678,0.0719,-11908.1685
C00682=51.936,84.362,71.920,178.6067,1.8290,-11911.6178
C00683=54.130,79.138,71.535,179.3164,4.6272,-11914.3719
C00684=53.356,73.536,71.060,-176.9938,6.7981,-11915.9638
C00685=49.842,68.316,70.157,-175.7735,6.1039,-11916.1137
C00686=45.816,62.906,68.324,-176.4873,5.0494,-11916.0668
C00687=42.239,58.063,65.929,-177.6829,3.4831,-11916.0347
C00688=39.736,54.260,63.612,179.8766,-0.2159,-11916.2163
C00689=39.035,51.313,61.945,-176.2551,-25.2833,-11917.2611
C00690=40.942,48.532,61.285,-153.9166,-28.7991,-11920.1513
C00691=43.085,46.550,61.257,-150.8922,-26.9372,-11922.7862
C00692=44.848,44.848,61.276,-151.9501,-28.0492,-11925.0000
C00693=46.550,43.085,61.257,-153.0632,-29.1083,-11927.2138
C00694=48.532,40.942,61.285,-151.1999,-26.0813,-11929.8487
C00695=51.313,39.035,61.945,-154.7168,-3.7449,-11932.7389
C00696=54.260,39.736,63.612,-179.7841,0.1234,-11933.7837
C00697=58.063,42.239,65.929,176.5169,-2.3171,-11933.9653
C00698=62.906,45.816,68.324,174.9506,-3.5127,-11933.9332
C00699=68.316,49.842,70.157,173.8961,-4.2265,-11933.8863
C00700=73.536,53.356,71.060,173.2019,-3.0062,-11934.0362
C00701=79.138,54.130,71.535,175.3728,0.6836,-11935.6281
C00702=84.362,51.936,71.920,178.1710,1.3933,-11938.3822
C00703=88.127,47.191,72.309,179.9281,0.1322,-11941.8315
C00704=91.053,41.335,72.565,179.9926,0.0163,-11945.5835
C00705=93.612,35.156,72.565,179.9938,0.0167,-11949.4163
C00706=95.684,28.946,72.309,179.9574,0.1443,-11953.1686
C00707=96.378,22.929,71.920,-179.6917,2.2779,-11956.6177
C00708=94.235,17.683,71.535,-177.2066,3.7570,-11959.3722
C00709=89.726,14.270,71.060,-173.0765,2.7000,-11960.9634
C00710=83.550,13.063,70.157,-172.7130,1.3383,-11961.1138
C00711=76.878,12.084,68.324,-173.9558,1.0926,-11961.0671
C00712=70.924,11.189,65.929,-175.9017,0.8265,-11961.0349
C00713=66.465,10.270,63.612,179.7601,-0.0654,-11961.2163
C00714=63.886,8.682,61.945,163.9488,-20.8208,-11962.2610
C00715=63.268,5.367,61.285,177.5626,-36.3112,-11965.1512
C00716=63.381,2.450,61.257,-178.0307,-36.9801,-11967.7863
C00717=63.425,0.000,61.276,-179.9993,-36.9988,-11970.0000
C00718=63.381,-2.450,61.257,178.0299,-36.9802,-11972.2137
C00719=63.268,-5.367,61.285,-177.5598,-36.3106,-11974.8488
C00720=63.886,-8.682,61.945,-163.9488,-20.8207,-11977.7390
C00721=66.465,-10.270,63.612,-179.7601,-0.0654,-11978.7837
C00722=70.924,-11.189,65.929,175.9017,0.8265,-11978.9651
C00723=76.878,-12.084,68.324,173.9558,1.0926,-11978.9329
C00724=83.550,-13.063,70.157,172.7130,1.3383,-11978.8862
C00725=89.726,-14.270,71.060,173.0765,2.7000,-11979.0366
C00726=94.235,-17.683,71.535,177.2066,3.7570,-11980.6278
C00727=96.378,-22.929,71.920,179.6917,2.2779,-11983.3823
C00728=95.684,-28.946,72.309,-179.9574,0.1443,-11986.8314
C00729=93.612,-35.156,72.565,-179.9938,0.0167,-11990.5837
C00730=91.053,-41.335,72.565,-179.9926,0.0163,-11994.4165
C00731=88.127,-47.191,72.309,-179.9281,0.1322,-11998.1685
C00732=84.362,-51.936,71.920,-178.1710,1.3933,-12001.6178
C00733=79.138,-54.130,71.535,-175.3728,0.6836,-12004.3719
C00734=73.536,-53.356,71.060,-173.2019,-3.0062,-12005.9638
C00735=68.316,-49.842,70.157,-173.8961,-4.2265,-12006.1137
C00736=62.906,-45.816,68.324,-174.9506,-3.5127,-12006.0668
C00737=58.063,-42.239,65.929,-176.5169,-2.3171,-12006.0347
C00738=54.260,-39.736,63.612,179.7841,0.1234,-12006.2163
C00739=51.313,-39.035,61.945,154.7167,-3.7449,-12007.2611
C00740=48.532,-40.942,61.285,151.2009,-26.0834,-12010.1513
C00741=46.550,-43.085,61.257,153.0628,-29.1078,-12012.7862
C00742=44.848,-44.848,61.276,151.9508,-28.0499,-12015.0000
C00743=43.085,-46.550,61.257,150.8917,-26.9368,-12017.2138
C00744=40.942,-48.532,61.285,153.9187,-28.8001,-12019.8487
C00745=39.035,-51.313,61.945,176.2551,-25.2832,-12022.7389
C00746=39.736,-54.260,63.612,-179.8766,-0.2159,-12023.7837
C00747=42.239,-58.063,65.929,177.6829,3.4831,-12023.9653
C00748=45.816,-62.906,68.324,176.4873,5.0494,-12023.9332
C00749=49.842,-68.316,70.157,175.7735,6.1039,-12023.8863
C00750=53.356,-73.536,71.060,176.9938,6.7981,-12024.0362
C00751=54.130,-79.138,71.535,-179.3164,4.6272,-12025.6281
C00752=51.936,-84.362,71.920,-178.6067,1.8290,-12028.3822
C00753=47.191,-88.127,72.309,-179.8678,0.0719,-12031.8315
C00754=41.335,-91.053,72.565,-179.9837,0.0074,-12035.5835
C00755=35.156,-93.612,72.565,-179.9833,0.0062,-12039.4163
C00756=28.946,-95.684,72.309,-179.8557,0.0426,-12043.1686
C00757=22.929,-96.378,71.920,-177.7221,-0.3083,-12046.6177
C00758=17.683,-94.235,71.535,-176.2430,-2.7934,-12049.3722
C00759=14.270,-89.726,71.060,-177.3000,-6.9235,-12050.9634
C00760=13.063,-83.550,70.157,-178.6617,-7.2870,-12051.1138
C00761=12.084,-76.878,68.324,-178.9074,-6.0442,-12051.0671
C00762=11.189,-70.924,65.929,-179.1735,-4.0983,-12051.0349
C00763=10.270,-66.465,63.612,179.9346,0.2399,-12051.2163
C00764=8.682,-63.886,61.945,159.1792,16.0512,-12052.2610
C00765=5.367,-63.268,61.285,143.6888,2.4374,-12055.1512
C00766=2.450,-63.381,61.257,143.0199,-1.9693,-12057.7863
C00767=0.000,-63.425,61.276,143.0012,-0.0007,-12060.0000
C00768=0.000,-63.425,61.276,143.0012,-0.0007,-12060.0000
C00769=-2.450,-63.381,61.257,143.0198,1.9701,-12062.2137
C00770=-5.367,-63.268,61.285,143.6894,-2.4402,-12064.8488
C00771=-8.682,-63.886,61.945,159.1793,-16.0512,-12067.7390
C00772=-10.270,-66.465,63.612,179.9346,-0.2399,-12068.7837
C00773=-11.189,-70.924,65.929,-179.1735,4.0983,-12068.9651
C00774=-12.084,-76.878,68.324,-178.9074,6.0442,-12068.9329
C00775=-13.063,-83.550,70.157,-178.6617,7.2870,-12068.8862
C00776=-14.270,-89.726,71.060,-177.3000,6.9235,-12069.0366
C00777=-17.683,-94.235,71.535,-176.2430,2.7934,-12070.6278
C00778=-22.929,-96.378,71.920,-177.7221,0.3083,-12073.3823
C00779=-28.946,-95.684,72.309,-179.8557,-0.0426,-12076.8314
C00780=-35.156,-93.612,72.565,-179.9833,-0.0062,-12080.5837
C00781=-41.335,-91.053,72.565,-179.9837,-0.0074,-12084.4165
C00782=-47.191,-88.127,72.309,-179.8678,-0.0719,-12088.1685
C00783=-51.936,-84.362,71.920,-178.6067,-1.8290,-12091.6178
C00784=-54.130,-79.138,71.535,-179.3164,-4.6272,-12094.3719
C00785=-53.356,-73.536,71.060,176.9938,-6.7981,-12095.9638
C00786=-49.842,-68.316,70.157,175.7735,-6.1039,-12096.1137
C00787=-45.816,-62.906,68.324,176.4873,-5.0494,-12096.0668
C00788=-42.239,-58.063,65.929,177.6829,-3.4831,-12096.0347
C00789=-39.736,-54.260,63.612,-179.8766,0.2159,-12096.2163
C00790=-39.035,-51.313,61.945,176.2551,25.2833,-12097.2611
C00791=-40.942,-48.532,61.285,153.9166,28.7991,-12100.1513
C00792=-43.085,-46.550,61.257,150.8922,26.9372,-12102.7862
C00793=-44.848,-44.848,61.276,151.9501,28.0492,-12105.0000
C00794=-46.550,-43.085,61.257,153.0632,29.1083,-12107.2138
C00795=-48.532,-40.942,61.285,151.1999,26.0813,-12109.8487
C00796=-51.313,-39.035,61.945,154.7168,3.7449,-12112.7389
C00797=-54.260,-39.736,63.612,179.7841,-0.1234,-12113.7837
C00798=-58.063,-42.239,65.929,-176.5169,2.3171,-12113.9653
C00799=-62.906,-45.816,68.324,-174.9506,3.5127,-12113.9332
C00800=-68.316,-49.842,70.157,-173.8961,4.2265,-12113.8863
C00801=-73.536,-53.356,71.060,-173.2019,3.0062,-12114.0362
C00802=-79.138,-54.130,71.535,-175.3728,-0.6836,-12115.6281
C00803=-84.362,-51.936,71.920,-178.1710,-1.3933,-12118.3822
C00804=-88.127,-47.191,72.309,-179.9281,-0.1322,-12121.8315
C00805=-91.053,-41.335,72.565,-179.9926,-0.0163,-12125.5835
C00806=-93.612,-35.156,72.565,-179.9938,-0.0167,-12129.4163
C00807=-95.684,-28.946,72.309,-179.9574,-0.1443,-12133.1686
C00808=-96.378,-22.929,71.920,179.6917,-2.2779,-12136.6177
C00809=-94.235,-17.683,71.535,177.2066,-3.7570,-12139.3722
C00810=-89.726,-14.270,71.060,173.0765,-2.7000,-12140.9634
C00811=-83.550,-13.063,70.157,172.7130,-1.3383,-12141.1138
C00812=-76.878,-12.084,68.324,173.9558,-1.0926,-12141.0671
C00813=-70.924,-11.189,65.929,175.9017,-0.8265,-12141.0349
C00814=-66.465,-10.270,63.612,-179.7601,0.0654,-12141.2163
C00815=-63.886,-8.682,61.945,-163.9488,20.8208,-12142.2610
C00816=-63.268,-5.367,61.285,-177.5626,36.3112,-12145.1512
C00817=-63.381,-2.450,61.257,178.0307,36.9801,-12147.7863
C00818=-63.425,0.000,61.276,179.9993,36.9988,-12150.0000
C00819=-63.381,2.450,61.257,-178.0299,36.9802,-12152.2137
C00820=-63.268,5.367,61.285,177.5598,36.3106,-12154.8488
C00821=-63.886,8.682,61.945,163.9488,20.8207,-12157.7390
C00822=-66.465,10.270,63.612,179.7601,0.0654,-12158.7837
C00823=-70.924,11.189,65.929,-175.9017,-0.8265,-12158.9651
C00824=-76.878,12.084,68.324,-173.9558,-1.0926,-12158.9329
C00825=-83.550,13.063,70.157,-172.7130,-1.3383,-12158.8862
C00826=-89.726,14.270,71.060,-173.0765,-2.7000,-12159.0366
C00827=-94.235,17.683,71.535,-177.2066,-3.7570,-12160.6278
C00828=-96.378,22.929,71.920,-179.6917,-2.2779,-12163.3823
C00829=-95.684,28.946,72.309,179.9574,-0.1443,-12166.8314
C00830=-93.612,35.156,72.565,179.9938,-0.0167,-12170.5837
C00831=-91.053,41.335,72.565,179.9926,-0.0163,-12174.4165
C00832=-88.127,47.191,72.309,179.9281,-0.1322,-12178.1685
C00833=-84.362,51.936,71.920,178.1710,-1.3933,-12181.6178
C00834=-79.138,54.130,71.535,175.3728,-0.6836,-12184.3719
C00835=-73.536,53.356,71.060,173.2019,3.0062,-12185.9638
C00836=-68.316,49.842,70.157,173.8961,4.2265,-12186.1137
C00837=-62.906,45.816,68.324,174.9506,3.5127,-12186.0668
C00838=-58.063,42.239,65.929,176.5169,2.3171,-12186.0347
C00839=-54.260,39.736,63.612,-179.7841,-0.1234,-12186.2163
C00840=-51.313,39.035,61.945,-154.7167,3.7449,-12187.2611
C00841=-48.532,40.942,61.285,-151.2009,26.0834,-12190.1513
C00842=-46.550,43.085,61.257,-153.0628,29.1078,-12192.7862
C00843=-44.848,44.848,61.276,-151.9508,28.0499,-12195.0000
C00844=-43.085,46.550,61.257,-150.8917,26.9368,-12197.2138
C00845=-40.942,48.532,61.285,-153.9187,28.8001,-12199.8487
C00846=-39.035,51.313,61.945,-176.2551,25.2832,-12202.7389
C00847=-39.736,54.260,63.612,179.8766,0.2159,-12203.7837
C00848=-42.239,58.063,65.929,-177.6829,-3.4831,-12203.9653
C00849=-45.816,62.906,68.324,-176.4873,-5.0494,-12203.9332
C00850=-49.842,68.316,70.157,-175.7735,-6.1039,-12203.8863
C00851=-53.356,73.536,71.060,-176.9938,-6.7981,-12204.0362
C00852=-54.130,79.138,71.535,179.3164,-4.6272,-12205.6281
C00853=-51.936,84.362,71.920,178.6067,-1.8290,-12208.3822
C00854=-47.191,88.127,72.309,179.8678,-0.0719,-12211.8315
C00855=-41.335,91.053,72.565,179.9837,-0.0074,-12215.5835
C00856=-35.156,93.612,72.565,179.9833,-0.0062,-12219.4163
C00857=-28.946,95.684,72.309,179.8557,-0.0426,-12223.1686
C00858=-22.929,96.378,71.920,177.7221,0.3083,-12226.6177
C00859=-17.683,94.235,71.535,176.2430,2.7934,-12229.3722
C00860=-14.270,89.726,71.060,177.3000,6.9235,-12230.9634
C00861=-13.063,83.550,70.157,178.6617,7.2870,-12231.1138
C00862=-12.084,76.878,68.324,178.9074,6.0442,-12231.0671
C00863=-11.189,70.924,65.929,179.1735,4.0983,-12231.0349
C00864=-10.270,66.465,63.612,-179.9346,-0.2399,-12231.2163
C00865=-8.682,63.886,61.945,-159.1793,-16.0512,-12232.2610
C00866=-5.367,63.268,61.285,-143.6894,-2.4402,-12235.1512
C00867=-2.450,63.381,61.257,-143.0198,1.9701,-12237.7863
C00868=0.000,63.425,61.276,-143.0012,-0.0007,-12240.0000
C00869=0.000,62.111,63.041,-143.6741,-0.0008,-12240.0000
C00870=2.330,62.072,63.021,-143.6912,-1.8775,-12242.1497
C00871=5.165,61.970,63.050,-144.4274,2.7476,-12244.7644
C00872=8.436,62.639,63.741,-160.6258,15.7082,-12247.6702
C00873=9.975,65.350,65.485,179.9114,-0.3487,-12248.6786
C00874=10.861,70.011,67.904,179.1939,-4.2042,-12248.8182
C00875=11.743,76.212,70.393,178.9773,-5.9076,-12248.7594
C00876=12.712,83.133,72.289,178.7756,-7.0021,-12248.6938
C00877=13.898,89.524,73.219,177.5056,-6.6475,-12248.8243
C00878=17.338,94.193,73.707,176.4305,-2.7219,-12250.4296
C00879=22.659,96.427,74.103,177.8254,-0.3086,-12253.2238
C00880=28.778,95.739,74.502,179.8617,0.0408,-12256.7302
C00881=35.099,93.634,74.765,179.9840,0.0060,-12260.5487
C00882=41.391,91.028,74.765,179.9845,0.0071,-12264.4516
C00883=47.349,88.047,74.502,179.8733,0.0690,-12268.2700
C00884=52.162,84.206,74.103,178.6800,1.7561,-12271.7764
C00885=54.344,78.865,73.707,179.3988,4.4445,-12274.5698
C00886=53.475,73.130,73.219,-177.0458,6.4591,-12276.1755
C00887=49.795,67.773,72.289,-175.8969,5.8218,-12276.3059
C00888=45.586,62.194,70.393,-176.5353,4.9034,-12276.2401
C00889=41.825,57.185,67.904,-177.5933,3.5437,-12276.1817
C00890=39.156,53.262,65.485,-179.8161,0.3093,-12276.3218
C00891=38.328,50.258,63.741,-177.1498,-24.1096,-12277.3300
C00892=40.167,47.472,63.050,-154.7424,-28.3541,-12280.2352
C00893=42.244,45.539,63.021,-151.5083,-26.4003,-12282.8504
C00894=43.919,43.919,63.041,-152.5290,-27.4701,-12285.0000
C00895=45.539,42.244,63.021,-153.6002,-28.4922,-12287.1496
C00896=47.472,40.167,63.050,-151.6449,-25.2554,-12289.7648
C00897=50.258,38.328,63.741,-155.8906,-2.8500,-12292.6700
C00898=53.262,39.156,65.485,179.6907,-0.1839,-12293.6782
C00899=57.185,41.825,67.904,176.4563,-2.4067,-12293.8183
C00900=62.194,45.586,70.393,175.0966,-3.4647,-12293.7599
C00901=67.773,49.795,72.289,174.1782,-4.1031,-12293.6941
C00902=73.130,53.475,73.219,173.5409,-2.9542,-12293.8245
C00903=78.865,54.344,73.707,175.5555,0.6012,-12295.4302
C00904=84.206,52.162,74.103,178.2439,1.3200,-12298.2236
C00905=88.047,47.349,74.502,179.9310,0.1267,-12301.7300
C00906=91.028,41.391,74.765,179.9929,0.0155,-12305.5484
C00907=93.634,35.099,74.765,179.9940,0.0160,-12309.4513
C00908=95.739,28.778,74.502,179.9592,0.1383,-12313.2698
C00909=96.427,22.659,74.103,-179.6914,2.1746,-12316.7762
C00910=94.193,17.338,73.707,-177.2781,3.5695,-12319.5704
C00911=89.524,13.898,73.219,-173.3525,2.4944,-12321.1757
C00912=83.133,12.712,72.289,-172.9979,1.2244,-12321.3062
C00913=76.212,11.743,70.393,-174.0924,1.0227,-12321.2406
C00914=70.011,10.861,67.904,-175.7958,0.8061,-12321.1818
C00915=65.350,9.975,65.485,-179.6513,0.0886,-12321.3214
C00916=62.639,8.436,63.741,164.2918,-19.3742,-12322.3298
C00917=61.970,5.165,63.050,177.2524,-35.5726,-12325.2356
C00918=62.072,2.330,63.021,-178.1225,-36.3088,-12327.8503
C00919=62.111,0.000,63.041,-179.9992,-36.3259,-12330.0000
C00920=62.072,-2.330,63.021,178.1217,-36.3088,-12332.1497
C00921=61.970,-5.165,63.050,-177.2496,-35.5720,-12334.7644
C00922=62.640,-8.436,63.741,-164.2918,-19.3740,-12337.6701
C00923=65.350,-9.975,65.485,179.6513,0.0886,-12338.6786
C00924=70.011,-10.861,67.904,175.7958,0.8061,-12338.8182
C00925=76.212,-11.743,70.393,174.0924,1.0227,-12338.7594
C00926=83.133,-12.712,72.289,172.9979,1.2244,-12338.6938
C00927=89.524,-13.898,73.219,173.3525,2.4944,-12338.8243
C00928=94.193,-17.338,73.707,177.2781,3.5695,-12340.4296
C00929=96.427,-22.659,74.103,179.6914,2.1746,-12343.2238
C00930=95.739,-28.778,74.502,-179.9592,0.1383,-12346.7302
C00931=93.634,-35.099,74.765,-179.9940,0.0160,-12350.5487
C00932=91.028,-41.391,74.765,-179.9929,0.0155,-12354.4516
C00933=88.047,-47.349,74.502,-179.9310,0.1267,-12358.2700
C00934=84.206,-52.162,74.103,-178.2439,1.3200,-12361.7764
C00935=78.865,-54.344,73.707,-175.5555,0.6012,-12364.5698
C00936=73.130,-53.475,73.219,-173.5409,-2.9542,-12366.1755
C00937=67.773,-49.795,72.289,-174.1782,-4.1031,-12366.3059
C00938=62.194,-45.586,70.393,-175.0966,-3.4647,-12366.2401
C00939=57.185,-41.825,67.904,-176.4563,-2.4067,-12366.1817
C00940=53.262,-39.156,65.485,-179.6907,-0.1839,-12366.3218
C00941=50.258,-38.328,63.741,155.8904,-2.8502,-12367.3300
C00942=47.472,-40.167,63.050,151.6459,-25.2576,-12370.2352
C00943=45.539,-42.244,63.021,153.5997,-28.4917,-12372.8504
C00944=43.919,-43.919,63.041,152.5299,-27.4710,-12375.0000
C00945=42.244,-45.539,63.021,151.5078,-26.3998,-12377.1496
C00946=40.167,-47.472,63.050,154.7446,-28.3551,-12379.7648
C00947=38.328,-50.258,63.741,177.1500,-24.1094,-12382.6700
C00948=39.156,-53.262,65.485,179.8161,0.3093,-12383.6782
C00949=41.825,-57.185,67.904,177.5933,3.5437,-12383.8183
C00950=45.586,-62.194,70.393,176.5353,4.9034,-12383.7599
C00951=49.795,-67.773,72.289,175.8969,5.8218,-12383.6941
C00952=53.475,-73.130,73.219,177.0458,6.4591,-12383.8245
C00953=54.344,-78.865,73.707,-179.3988,4.4445,-12385.4302
C00954=52.162,-84.206,74.103,-178.6800,1.7561,-12388.2236
C00955=47.349,-88.047,74.502,-179.8733,0.0690,-12391.7300
C00956=41.391,-91.028,74.765,-179.9845,0.0071,-12395.5484
C00957=35.099,-93.634,74.765,-179.9840,0.0060,-12399.4513
C00958=28.778,-95.739,74.502,-179.8617,0.0408,-12403.2698
C00959=22.659,-96.427,74.103,-177.8254,-0.3086,-12406.7762
C00960=17.338,-94.193,73.707,-176.4305,-2.7219,-12409.5704
C00961=13.898,-89.524,73.219,-177.5056,-6.6475,-12411.1757
C00962=12.712,-83.133,72.289,-178.7756,-7.0021,-12411.3062
C00963=11.743,-76.212,70.393,-178.9773,-5.9076,-12411.2406
C00964=10.861,-70.011,67.904,-179.1939,-4.2042,-12411.1818
C00965=9.975,-65.350,65.485,-179.9114,-0.3487,-12411.3214
C00966=8.436,-62.639,63.741,160.6258,15.7082,-12412.3298
C00967=5.165,-61.970,63.050,144.4274,2.7476,-12415.2356
C00968=2.330,-62.072,63.021,143.6912,-1.8775,-12417.8503
C00969=0.000,-62.111,63.041,143.6741,-0.0008,-12420.0000
C00970=0.000,-62.111,63.041,143.6741,-0.0008,-12420.0000
C00971=-2.330,-62.072,63.021,143.6912,1.8783,-12422.1497
C00972=-5.165,-61.970,63.050,144.4280,-2.7504,-12424.7644
C00973=-8.436,-62.640,63.741,160.6260,-15.7082,-12427.6701
C00974=-9.975,-65.350,65.485,-179.9114,0.3487,-12428.6786
C00975=-10.861,-70.011,67.904,-179.1939,4.2042,-12428.8182
C00976=-11.743,-76.212,70.393,-178.9773,5.9076,-12428.7594
C00977=-12.712,-83.133,72.289,-178.7756,7.0021,-12428.6938
C00978=-13.898,-89.524,73.219,-177.5056,6.6475,-12428.8243
C00979=-17.338,-94.193,73.707,-176.4305,2.7219,-12430.4296
C00980=-22.659,-96.427,74.103,-177.8254,0.3086,-12433.2238
C00981=-28.778,-95.739,74.502,-179.8617,-0.0408,-12436.7302
C00982=-35.099,-93.634,74.765,-179.9840,-0.0060,-12440.5487
C00983=-41.391,-91.028,74.765,-179.9845,-0.0071,-12444.4516
C00984=-47.349,-88.047,74.502,-179.8733,-0.0690,-12448.2700
C00985=-52.162,-84.206,74.103,-178.6800,-1.7561,-12451.7764
C00986=-54.344,-78.865,73.707,-179.3988,-4.4445,-12454.5698
C00987=-53.475,-73.130,73.219,177.0458,-6.4591,-12456.1755
C00988=-49.795,-67.773,72.289,175.8969,-5.8218,-12456.3059
C00989=-45.586,-62.194,70.393,176.5353,-4.9034,-12456.2401
C00990=-41.825,-57.185,67.904,177.5933,-3.5437,-12456.1817
C00991=-39.156,-53.262,65.485,179.8161,-0.3093,-12456.3218
C00992=-38.328,-50.258,63.741,177.1498,24.1096,-12457.3300
C00993=-40.167,-47.472,63.050,154.7424,28.3541,-12460.2352
C00994=-42.244,-45.539,63.021,151.5083,26.4003,-12462.8504
C00995=-43.919,-43.919,63.041,152.5290,27.4701,-12465.0000
C00996=-45.539,-42.244,63.021,153.6002,28.4922,-12467.1496
C00997=-47.472,-40.167,63.050,151.6449,25.2554,-12469.7648
C00998=-50.258,-38.328,63.741,155.8906,2.8500,-12472.6700
C00999=-53.262,-39.156,65.485,-179.6907,0.1839,-12473.6782
C01000=-57.185,-41.825,67.904,-176.4563,2.4067,-12473.8183
C01001=-62.194,-45.586,70.393,-175.0966,3.4647,-12473.7599
C01002=-67.773,-49.795,72.289,-174.1782,4.1031,-12473.6941
C01003=-73.130,-53.475,73.219,-173.5409,2.9542,-12473.8245
C01004=-78.865,-54.344,73.707,-175.5555,-0.6012,-12475.4302
C01005=-84.206,-52.162,74.103,-178.2439,-1.3200,-12478.2236
C01006=-88.047,-47.349,74.502,-179.9310,-0.1267,-12481.7300
C01007=-91.028,-41.391,74.765,-179.9929,-0.0155,-12485.5484
C01008=-93.634,-35.099,74.765,-179.9940,-0.0160,-12489.4513
C01009=-95.739,-28.778,74.502,-179.9592,-0.1383,-12493.2698
C01010=-96.427,-22.659,74.103,179.6914,-2.1746,-12496.7762
C01011=-94.193,-17.338,73.707,177.2781,-3.5695,-12499.5704
C01012=-89.524,-13.898,73.219,173.3525,-2.4944,-12501.1757
C01013=-83.133,-12.712,72.289,172.9979,-1.2244,-12501.3062
C01014=-76.212,-11.743,70.393,174.0924,-1.0227,-12501.2406
C01015=-70.011,-10.861,67.904,175.7958,-0.8061,-12501.1818
C01016=-65.350,-9.975,65.485,179.6513,-0.0886,-12501.3214
C01017=-62.639,-8.436,63.741,-164.2918,19.3742,-12502.3298
C01018=-61.970,-5.165,63.050,-177.2524,35.5726,-12505.2356
C01019=-62.072,-2.330,63.021,178.1225,36.3088,-12507.8503
C01020=-62.111,0.000,63.041,179.9992,36.3259,-12510.0000
C01021=-62.072,2.330,63.021,-178.1217,36.3088,-12512.1497
C01022=-61.970,5.165,63.050,177.2496,35.5720,-12514.7644
C01023=-62.640,8.436,63.741,164.2918,19.3740,-12517.6701
C01024=-65.350,9.975,65.485,-179.6513,-0.0886,-12518.6786
C01025=-70.011,10.861,67.904,-175.7958,-0.8061,-12518.8182
C01026=-76.212,11.743,70.393,-174.0924,-1.0227,-12518.7594
C01027=-83.133,12.712,72.289,-172.9979,-1.2244,-12518.6938
C01028=-89.524,13.898,73.219,-173.3525,-2.4944,-12518.8243
C01029=-94.193,17.338,73.707,-177.2781,-3.5695,-12520.4296
C01030=-96.427,22.659,74.103,-179.6914,-2.1746,-12523.2238
C01031=-95.739,28.778,74.502,179.9592,-0.1383,-12526.7302
C01032=-93.634,35.099,74.765,179.9940,-0.0160,-12530.5487
C01033=-91.028,41.391,74.765,179.9929,-0.0155,-12534.4516
C01034=-88.047,47.349,74.502,179.9310,-0.1267,-12538.2700
C01035=-84.206,52.162,74.103,178.2439,-1.3200,-12541.7764
C01036=-78.865,54.344,73.707,175.5555,-0.6012,-12544.5698
C01037=-73.130,53.475,73.219,173.5409,2.9542,-12546.1755
C01038=-67.773,49.795,72.289,174.1782,4.1031,-12546.3059
C01039=-62.194,45.586,70.393,175.0966,3.4647,-12546.2401
C01040=-57.185,41.825,67.904,176.4563,2.4067,-12546.1817
C01041=-53.262,39.156,65.485,179.6907,0.1839,-12546.3218
C01042=-50.258,38.328,63.741,-155.8904,2.8502,-12547.3300
C01043=-47.472,40.167,63.050,-151.6459,25.2576,-12550.2352
C01044=-45.539,42.244,63.021,-153.5997,28.4917,-12552.8504
C01045=-43.919,43.919,63.041,-152.5299,27.4710,-12555.0000
C01046=-42.244,45.539,63.021,-151.5078,26.3998,-12557.1496
C01047=-40.167,47.472,63.050,-154.7446,28.3551,-12559.7648
C01048=-38.328,50.258,63.741,-177.1500,24.1094,-12562.6700
C01049=-39.156,53.262,65.485,-179.8161,-0.3093,-12563.6782
C01050=-41.825,57.185,67.904,-177.5933,-3.5437,-12563.8183
C01051=-45.586,62.194,70.393,-176.5353,-4.9034,-12563.7599
C01052=-49.795,67.773,72.289,-175.8969,-5.8218,-12563.6941
C01053=-53.475,73.130,73.219,-177.0458,-6.4591,-12563.8245
C01054=-54.344,78.865,73.707,179.3988,-4.4445,-12565.4302
C01055=-52.162,84.206,74.103,178.6800,-1.7561,-12568.2236
C01056=-47.349,88.047,74.502,179.8733,-0.0690,-12571.7300
C01057=-41.391,91.028,74.765,179.9845,-0.0071,-12575.5484
C01058=-35.099,93.634,74.765,179.9840,-0.0060,-12579.4513
C01059=-28.778,95.739,74.502,179.8617,-0.0408,-12583.2698
C01060=-22.659,96.427,74.103,177.8254,0.3086,-12586.7762
C01061=-17.338,94.193,73.707,176.4305,2.7219,-12589.5704
C01062=-13.898,89.524,73.219,177.5056,6.6475,-12591.1757
C01063=-12.712,83.133,72.289,178.7756,7.0021,-12591.3062
C01064=-11.743,76.212,70.393,178.9773,5.9076,-12591.2406
C01065=-10.861,70.011,67.904,179.1939,4.2042,-12591.1818
C01066=-9.975,65.350,65.485,179.9114,0.3487,-12591.3214
C01067=-8.436,62.640,63.741,-160.6260,-15.7082,-12592.3299
C01068=-5.165,61.970,63.050,-144.4280,-2.7504,-12595.2356
C01069=-2.330,62.072,63.021,-143.6912,1.8783,-12597.8503
C01070=0.000,62.111,63.041,-143.6741,-0.0008,-12600.0000
C01071=0.000,60.820,64.822,-144.4513,-0.0008,-12600.0000
C01072=2.212,60.785,64.801,-144.4668,-1.7783,-12602.0841
C01073=4.967,60.695,64.832,-145.2737,3.0327,-12604.6784
C01074=8.195,61.417,65.554,-162.0706,15.2576,-12607.6002
C01075=9.686,64.262,67.375,179.7975,-0.8529,-12608.5715
C01076=10.544,69.129,69.894,179.2239,-4.2461,-12608.6723
C01077=11.418,75.576,72.474,179.0505,-5.7116,-12608.5913
C01078=12.382,82.740,74.428,178.8887,-6.6531,-12608.5111
C01079=13.550,89.334,75.383,177.7173,-6.3021,-12608.6248
C01080=17.016,94.154,75.883,176.6505,-2.6124,-12610.2442
C01081=22.407,96.473,76.288,177.9510,-0.3030,-12613.0758
C01082=28.621,95.791,76.696,179.8693,0.0384,-12616.6354
C01083=35.046,93.654,76.964,179.9850,0.0056,-12620.5162
C01084=41.442,91.005,76.964,179.9854,0.0067,-12624.4836
C01085=47.497,87.973,76.696,179.8804,0.0653,-12628.3648
C01086=52.372,84.060,76.288,178.7650,1.6633,-12631.9242
C01087=54.545,78.609,75.883,179.4774,4.2121,-12634.7559
C01088=53.588,72.750,75.383,-177.1430,6.0665,-12636.3755
C01089=49.751,67.261,74.428,-176.0664,5.4947,-12636.4893
C01090=45.367,61.514,72.474,-176.6232,4.7129,-12636.4090
C01091=41.426,56.337,69.894,-177.5424,3.5522,-12636.3280
C01092=38.591,52.289,67.375,-179.5401,0.7463,-12636.4285
C01093=37.634,49.223,65.554,-177.9435,-22.8637,-12637.4001
C01094=39.406,46.429,64.832,-155.6464,-27.8147,-12640.3225
C01095=41.417,44.545,64.801,-152.2131,-25.7824,-12642.9160
C01096=43.006,43.006,64.822,-153.1928,-26.8062,-12645.0000
C01097=44.545,41.417,64.801,-154.2181,-27.7874,-12647.0840
C01098=46.430,39.405,64.832,-152.1844,-24.3513,-12649.6788
C01099=49.223,37.634,65.554,-157.1366,-2.0563,-12652.5999
C01100=52.289,38.591,67.375,179.2537,-0.4599,-12653.5715
C01101=56.337,41.426,69.894,176.4478,-2.4576,-12653.6720
C01102=61.514,45.367,72.474,175.2871,-3.3768,-12653.5910
C01103=67.261,49.751,74.428,174.5053,-3.9336,-12653.5107
C01104=72.750,53.588,75.383,173.9335,-2.8570,-12653.6245
C01105=78.609,54.545,75.883,175.7879,0.5226,-12655.2441
C01106=84.060,52.372,76.288,178.3367,1.2350,-12658.0758
C01107=87.973,47.497,76.696,179.9347,0.1196,-12661.6352
C01108=91.005,41.442,76.964,179.9933,0.0146,-12665.5164
C01109=93.654,35.046,76.964,179.9944,0.0150,-12669.4838
C01110=95.791,28.621,76.696,179.9616,0.1307,-12673.3646
C01111=96.473,22.407,76.288,-179.6970,2.0490,-12676.9242
C01112=94.154,17.016,75.883,-177.3876,3.3495,-12679.7558
C01113=89.334,13.550,75.383,-173.6979,2.2827,-12681.3752
C01114=82.740,12.382,74.428,-173.3469,1.1113,-12681.4889
C01115=75.576,11.418,72.474,-174.2884,0.9495,-12681.4087
C01116=69.129,10.544,69.894,-175.7539,0.7761,-12681.3277
C01117=64.262,9.686,67.375,-179.1471,0.2025,-12681.4285
C01118=61.417,8.195,65.554,164.7424,-17.9294,-12682.3998
C01119=60.695,4.967,64.832,176.9673,-34.7263,-12685.3216
C01120=60.785,2.212,64.801,-178.2217,-35.5332,-12687.9159
C01121=60.820,0.000,64.822,-179.9992,-35.5487,-12690.0000
C01122=60.785,-2.212,64.801,178.2207,-35.5333,-12692.0841
C01123=60.695,-4.967,64.832,-176.9646,-34.7257,-12694.6784
C01124=61.417,-8.195,65.554,-164.7424,-17.9290,-12697.6002
C01125=64.262,-9.686,67.375,179.1471,0.2025,-12698.5715
C01126=69.129,-10.544,69.894,175.7539,0.7761,-12698.6723
C01127=75.576,-11.418,72.474,174.2884,0.9495,-12698.5913
C01128=82.740,-12.382,74.428,173.3469,1.1113,-12698.5111
C01129=89.334,-13.550,75.383,173.6979,2.2827,-12698.6248
C01130=94.154,-17.016,75.883,177.3876,3.3495,-12700.2442
C01131=96.473,-22.407,76.288,179.6970,2.0490,-12703.0758
C01132=95.791,-28.621,76.696,-179.9616,0.1307,-12706.6354
C01133=93.654,-35.046,76.964,-179.9944,0.0150,-12710.5162
C01134=91.005,-41.442,76.964,-179.9933,0.0146,-12714.4836
C01135=87.973,-47.497,76.696,-179.9347,0.1196,-12718.3648
C01136=84.060,-52.372,76.288,-178.3367,1.2350,-12721.9242
C01137=78.609,-54.545,75.883,-175.7879,0.5226,-12724.7559
C01138=72.750,-53.588,75.383,-173.9335,-2.8570,-12726.3755
C01139=67.261,-49.751,74.428,-174.5053,-3.9336,-12726.4893
C01140=61.514,-45.367,72.474,-175.2871,-3.3768,-12726.4090
C01141=56.337,-41.426,69.894,-176.4478,-2.4576,-12726.3280
C01142=52.289,-38.591,67.375,-179.2537,-0.4599,-12726.4285
C01143=49.223,-37.634,65.554,157.1363,-2.0565,-12727.4001
C01144=46.429,-39.406,64.832,152.1853,-24.3536,-12730.3225
C01145=44.545,-41.417,64.801,154.2176,-27.7869,-12732.9160
C01146=43.006,-43.006,64.822,153.1938,-26.8072,-12735.0000
C01147=41.417,-44.545,64.801,152.2126,-25.7819,-12737.0840
C01148=39.405,-46.430,64.832,155.6487,-27.8156,-12739.6788
C01149=37.634,-49.223,65.554,177.9437,-22.8634,-12742.5999
C01150=38.591,-52.289,67.375,179.5401,0.7463,-12743.5715
C01151=41.426,-56.337,69.894,177.5424,3.5522,-12743.6720
C01152=45.367,-61.514,72.474,176.6232,4.7129,-12743.5910
C01153=49.751,-67.261,74.428,176.0664,5.4947,-12743.5107
C01154=53.588,-72.750,75.383,177.1430,6.0665,-12743.6245
C01155=54.545,-78.609,75.883,-179.4774,4.2121,-12745.2441
C01156=52.372,-84.060,76.288,-178.7650,1.6633,-12748.0758
C01157=47.497,-87.973,76.696,-179.8804,0.0653,-12751.6352
C01158=41.442,-91.005,76.964,-179.9854,0.0067,-12755.5164
C01159=35.046,-93.654,76.964,-179.9850,0.0056,-12759.4838
C01160=28.621,-95.791,76.696,-179.8693,0.0384,-12763.3646
C01161=22.407,-96.473,76.288,-177.9510,-0.3030,-12766.9242
C01162=17.016,-94.154,75.883,-176.6505,-2.6124,-12769.7558
C01163=13.550,-89.334,75.383,-177.7173,-6.3021,-12771.3752
C01164=12.382,-82.740,74.428,-178.8887,-6.6531,-12771.4889
C01165=11.418,-75.576,72.474,-179.0505,-5.7116,-12771.4087
C01166=10.544,-69.129,69.894,-179.2239,-4.2461,-12771.3277
C01167=9.686,-64.262,67.375,-179.7975,-0.8529,-12771.4285
C01168=8.195,-61.417,65.554,162.0706,15.2576,-12772.3998
C01169=4.967,-60.695,64.832,145.2737,3.0327,-12775.3216
C01170=2.212,-60.785,64.801,144.4668,-1.7783,-12777.9159
C01171=0.000,-60.820,64.822,144.4513,-0.0008,-12780.0000
C01172=0.000,-60.820,64.822,144.4513,-0.0008,-12780.0000
C01173=-2.212,-60.785,64.801,144.4667,1.7793,-12782.0841
C01174=-4.967,-60.695,64.832,145.2743,-3.0354,-12784.6784
C01175=-8.195,-61.417,65.554,162.0710,-15.2576,-12787.6002
C01176=-9.686,-64.262,67.375,-179.7975,0.8529,-12788.5715
C01177=-10.544,-69.129,69.894,-179.2239,4.2461,-12788.6723
C01178=-11.418,-75.576,72.474,-179.0505,5.7116,-12788.5913
C01179=-12.382,-82.740,74.428,-178.8887,6.6531,-12788.5111
C01180=-13.550,-89.334,75.383,-177.7173,6.3021,-12788.6248
C01181=-17.016,-94.154,75.883,-176.6505,2.6124,-12790.2442
C01182=-22.407,-96.473,76.288,-177.9510,0.3030,-12793.0758
C01183=-28.621,-95.791,76.696,-179.8693,-0.0384,-12796.6354
C01184=-35.046,-93.654,76.964,-179.9850,-0.0056,-12800.5162
C01185=-41.442,-91.005,76.964,-179.9854,-0.0067,-12804.4836
C01186=-47.497,-87.973,76.696,-179.8804,-0.0653,-12808.3648
C01187=-52.372,-84.060,76.288,-178.7650,-1.6633,-12811.9242
C01188=-54.545,-78.609,75.883,-179.4774,-4.2121,-12814.7559
C01189=-53.588,-72.750,75.383,177.1430,-6.0665,-12816.3755
C01190=-49.751,-67.261,74.428,176.0664,-5.4947,-12816.4893
C01191=-45.367,-61.514,72.474,176.6232,-4.7129,-12816.4090
C01192=-41.426,-56.337,69.894,177.5424,-3.5522,-12816.3280
C01193=-38.591,-52.289,67.375,179.5401,-0.7463,-12816.4285
C01194=-37.634,-49.223,65.554,177.9435,22.8637,-12817.4001
C01195=-39.406,-46.429,64.832,155.6464,27.8147,-12820.3225
C01196=-41.417,-44.545,64.801,152.2131,25.7824,-12822.9160
C01197=-43.006,-43.006,64.822,153.1928,26.8062,-12825.0000
C01198=-44.545,-41.417,64.801,154.2181,27.7874,-12827.0840
C01199=-46.430,-39.405,64.832,152.1844,24.3513,-12829.6788
C01200=-49.223,-37.634,65.554,157.1366,2.0563,-12832.5999
C01201=-52.289,-38.591,67.375,-179.2537,0.4599,-12833.5715
C01202=-56.337,-41.426,69.894,-176.4478,2.4576,-12833.6720
C01203=-61.514,-45.367,72.474,-175.2871,3.3768,-12833.5910
C01204=-67.261,-49.751,74.428,-174.5053,3.9336,-12833.5107
C01205=-72.750,-53.588,75.383,-173.9335,2.8570,-12833.6245
C01206=-78.609,-54.545,75.883,-175.7879,-0.5226,-12835.2441
C01207=-84.060,-52.372,76.288,-178.3367,-1.2350,-12838.0758
C01208=-87.973,-47.497,76.696,-179.9347,-0.1196,-12841.6352
C01209=-91.005,-41.442,76.964,-179.9933,-0.0146,-12845.5164
C01210=-93.654,-35.046,76.964,-179.9944,-0.0150,-12849.4838
C01211=-95.791,-28.621,76.696,-179.9616,-0.1307,-12853.3646
C01212=-96.473,-22.407,76.288,179.6970,-2.0490,-12856.9242
C01213=-94.154,-17.016,75.883,177.3876,-3.3495,-12859.7558
C01214=-89.334,-13.550,75.383,173.6979,-2.2827,-12861.3752
C01215=-82.740,-12.382,74.428,173.3469,-1.1113,-12861.4889
C01216=-75.576,-11.418,72.474,174.2884,-0.9495,-12861.4087
C01217=-69.129,-10.544,69.894,175.7539,-0.7761,-12861.3277
C01218=-64.262,-9.686,67.375,179.1471,-0.2025,-12861.4285
C01219=-61.417,-8.195,65.554,-164.7424,17.9294,-12862.3998
C01220=-60.695,-4.967,64.832,-176.9673,34.7263,-12865.3216
C01221=-60.785,-2.212,64.801,178.2217,35.5332,-12867.9159
C01222=-60.820,0.000,64.822,179.9992,35.5487,-12870.0000
C01223=-60.785,2.212,64.801,-178.2207,35.5333,-12872.0841
C01224=-60.695,4.967,64.832,176.9646,34.7257,-12874.6784
C01225=-61.417,8.195,65.554,164.7424,17.9290,-12877.6002
C01226=-64.262,9.686,67.375,-179.1471,-0.2025,-12878.5715
C01227=-69.129,10.544,69.894,-175.7539,-0.7761,-12878.6723
C01228=-75.576,11.418,72.474,-174.2884,-0.9495,-12878.5913
C01229=-82.740,12.382,74.428,-173.3469,-1.1113,-12878.5111
C01230=-89.334,13.550,75.383,-173.6979,-2.2827,-12878.6248
C01231=-94.154,17.016,75.883,-177.3876,-3.3495,-12880.2442
C01232=-96.473,22.407,76.288,-179.6970,-2.0490,-12883.0758
C01233=-95.791,28.621,76.696,179.9616,-0.1307,-12886.6354
C01234=-93.654,35.046,76.964,179.9944,-0.0150,-12890.5162
C01235=-91.005,41.442,76.964,179.9933,-0.0146,-12894.4836
C01236=-87.973,47.497,76.696,179.9347,-0.1196,-12898.3648
C01237=-84.060,52.372,76.288,178.3367,-1.2350,-12901.9242
C01238=-78.609,54.545,75.883,175.7879,-0.5226,-12904.7559
C01239=-72.750,53.588,75.383,173.9335,2.8570,-12906.3755
C01240=-67.261,49.751,74.428,174.5053,3.9336,-12906.4893
C01241=-61.514,45.367,72.474,175.2871,3.3768,-12906.4090
C01242=-56.337,41.426,69.894,176.4478,2.4576,-12906.3280
C01243=-52.289,38.591,67.375,179.2537,0.4599,-12906.4285
C01244=-49.223,37.634,65.554,-157.1363,2.0565,-12907.4001
C01245=-46.429,39.406,64.832,-152.1853,24.3536,-12910.3225
C01246=-44.545,41.417,64.801,-154.2176,27.7869,-12912.9160
C01247=-43.006,43.006,64.822,-153.1938,26.8072,-12915.0000
C01248=-41.417,44.545,64.801,-152.2126,25.7819,-12917.0840
C01249=-39.405,46.430,64.832,-155.6487,27.8156,-12919.6788
C01250=-37.634,49.223,65.554,-177.9437,22.8634,-12922.5999
C01251=-38.591,52.289,67.375,-179.5401,-0.7463,-12923.5715
C01252=-41.426,56.337,69.894,-177.5424,-3.5522,-12923.6720
C01253=-45.367,61.514,72.474,-176.6232,-4.7129,-12923.5910
C01254=-49.751,67.261,74.428,-176.0664,-5.4947,-12923.5107
C01255=-53.588,72.750,75.383,-177.1430,-6.0665,-12923.6245
C01256=-54.545,78.609,75.883,179.4774,-4.2121,-12925.2441
C01257=-52.372,84.060,76.288,178.7650,-1.6633,-12928.0758
C01258=-47.497,87.973,76.696,179.8804,-0.0653,-12931.6352
C01259=-41.442,91.005,76.964,179.9854,-0.0067,-12935.5164
C01260=-35.046,93.654,76.964,179.9850,-0.0056,-12939.4838
C01261=-28.621,95.791,76.696,179.8693,-0.0384,-12943.3646
C01262=-22.407,96.473,76.288,177.9510,0.3030,-12946.9242
C01263=-17.016,94.154,75.883,176.6505,2.6124,-12949.7558
C01264=-13.550,89.334,75.383,177.7173,6.3021,-12951.3752
C01265=-12.382,82.740,74.428,178.8887,6.6531,-12951.4889
C01266=-11.418,75.576,72.474,179.0505,5.7116,-12951.4087
C01267=-10.544,69.129,69.894,179.2239,4.2461,-12951.3277
C01268=-9.686,64.262,67.375,179.7975,0.8529,-12951.4285
C01269=-8.195,61.417,65.554,-162.0710,-15.2576,-12952.3998
C01270=-4.967,60.695,64.832,-145.2743,-3.0354,-12955.3216
C01271=-2.212,60.785,64.801,-144.4667,1.7793,-12957.9159
C01272=0.000,60.820,64.822,-144.4513,-0.0008,-12960.0000
C01273=0.000,59.554,66.621,-145.3415,-0.0009,-12960.0000
C01274=2.097,59.523,66.599,-145.3553,-1.6722,-12962.0177
C01275=4.772,59.445,66.632,-146.2352,3.2869,-12964.5896
C01276=7.959,60.221,67.386,-163.5021,14.7072,-12967.5288
C01277=9.406,63.206,69.285,179.7171,-1.2730,-12968.4644
C01278=10.239,68.282,71.901,179.2620,-4.2251,-12968.5281
C01279=11.109,74.974,74.567,179.1263,-5.4571,-12968.4283
C01280=12.073,82.372,76.575,179.0007,-6.2410,-12968.3383
C01281=13.226,89.158,77.551,177.9343,-5.8891,-12968.4379
C01282=16.717,94.118,78.062,176.9018,-2.4653,-12970.0717
C01283=22.174,96.515,78.476,178.0988,-0.2913,-12972.9390
C01284=28.477,95.839,78.891,179.8785,0.0356,-12976.5485
C01285=34.998,93.673,79.163,179.9861,0.0052,-12980.4866
C01286=41.489,90.984,79.163,179.9865,0.0062,-12984.5131
C01287=47.632,87.904,78.891,179.8889,0.0607,-12988.4517
C01288=52.567,83.926,78.476,178.8613,1.5505,-12992.0609
C01289=54.731,78.373,78.062,179.5514,3.9310,-12994.9281
C01290=53.692,72.396,77.551,-177.2844,5.6222,-12996.5622
C01291=49.709,66.782,76.575,-176.2813,5.1235,-12996.6621
C01292=45.159,60.870,74.567,-176.7508,4.4791,-12996.5714
C01293=41.042,55.523,71.901,-177.5304,3.5105,-12996.4714
C01294=38.042,51.344,69.285,-179.2998,1.1002,-12996.5356
C01295=36.955,48.211,67.386,-178.6352,-21.5554,-12997.4711
C01296=38.660,45.408,66.632,-156.6295,-27.1736,-13000.4108
C01297=40.607,43.572,66.599,-153.0121,-25.0783,-13002.9827
C01298=42.111,42.111,66.621,-153.9470,-26.0519,-13005.0000
C01299=43.571,40.607,66.599,-154.9223,-26.9884,-13007.0166
C01300=45.409,38.659,66.632,-152.8255,-23.3682,-13009.5906
C01301=48.211,36.955,67.386,-158.4450,-1.3645,-13012.5289
C01302=51.344,38.042,69.285,178.8998,-0.7002,-13013.4644
C01303=55.523,41.042,71.901,176.4895,-2.4696,-13013.5286
C01304=60.870,45.159,74.567,175.5209,-3.2492,-13013.4286
C01305=66.782,49.709,76.575,174.8765,-3.7187,-13013.3379
C01306=72.396,53.692,77.551,174.3778,-2.7156,-13013.4378
C01307=78.373,54.731,78.062,176.0690,0.4486,-13015.0719
C01308=83.926,52.567,78.476,178.4495,1.1387,-13017.9391
C01309=87.904,47.632,78.891,179.9393,0.1111,-13021.5483
C01310=90.984,41.489,79.163,179.9938,0.0135,-13025.4869
C01311=93.673,34.998,79.163,179.9948,0.0139,-13029.5134
C01312=95.839,28.477,78.891,179.9644,0.1215,-13033.4515
C01313=96.515,22.174,78.476,-179.7087,1.9012,-13037.0610
C01314=94.118,16.717,78.062,-177.5347,3.0982,-13039.9283
C01315=89.158,13.226,77.551,-174.1109,2.0657,-13041.5621
C01316=82.372,12.073,76.575,-173.7590,0.9993,-13041.6617
C01317=74.974,11.109,74.567,-174.5429,0.8737,-13041.5717
C01318=68.282,10.239,71.901,-175.7749,0.7380,-13041.4719
C01319=63.206,9.406,69.285,-178.7270,0.2829,-13041.5356
C01320=60.221,7.959,67.386,165.2928,-16.4979,-13042.4712
C01321=59.445,4.772,66.632,176.7131,-33.7648,-13045.4104
C01322=59.523,2.097,66.599,-178.3278,-34.6447,-13047.9823
C01323=59.554,0.000,66.621,-179.9991,-34.6585,-13050.0000
C01324=59.523,-2.096,66.599,178.3268,-34.6448,-13052.0167
C01325=59.445,-4.772,66.632,-176.7103,-33.7640,-13054.5896
C01326=60.222,-7.959,67.386,-165.2928,-16.4975,-13057.5286
C01327=63.206,-9.406,69.285,178.7270,0.2829,-13058.4644
C01328=68.282,-10.239,71.901,175.7749,0.7380,-13058.5281
C01329=74.974,-11.109,74.567,174.5429,0.8737,-13058.4283
C01330=82.372,-12.073,76.575,173.7590,0.9993,-13058.3383
C01331=89.158,-13.226,77.551,174.1109,2.0657,-13058.4379
C01332=94.118,-16.717,78.062,177.5347,3.0982,-13060.0717
C01333=96.515,-22.174,78.476,179.7087,1.9012,-13062.9390
C01334=95.839,-28.477,78.891,-179.9644,0.1215,-13066.5485
C01335=93.673,-34.998,79.163,-179.9948,0.0139,-13070.4866
C01336=90.984,-41.489,79.163,-179.9938,0.0135,-13074.5131
C01337=87.904,-47.632,78.891,-179.9393,0.1111,-13078.4517
C01338=83.926,-52.567,78.476,-178.4495,1.1387,-13082.0609
C01339=78.373,-54.731,78.062,-176.0690,0.4486,-13084.9281
C01340=72.396,-53.692,77.551,-174.3778,-2.7156,-13086.5622
C01341=66.782,-49.709,76.575,-174.8765,-3.7187,-13086.6621
C01342=60.870,-45.159,74.567,-175.5209,-3.2492,-13086.5714
C01343=55.523,-41.042,71.901,-176.4895,-2.4696,-13086.4714
C01344=51.344,-38.042,69.285,-178.8998,-0.7002,-13086.5356
C01345=48.211,-36.955,67.386,158.4446,-1.3648,-13087.4711
C01346=45.408,-38.660,66.632,152.8264,-23.3705,-13090.4108
C01347=43.572,-40.607,66.599,154.9217,-26.9879,-13092.9827
C01348=42.111,-42.111,66.621,153.9481,-26.0530,-13095.0000
C01349=40.607,-43.571,66.599,153.0116,-25.0777,-13097.0166
C01350=38.659,-45.409,66.632,156.6318,-27.1745,-13099.5906
C01351=36.955,-48.211,67.386,178.6355,-21.5550,-13102.5289
C01352=38.042,-51.344,69.285,179.2998,1.1002,-13103.4644
C01353=41.042,-55.523,71.901,177.5304,3.5105,-13103.5286
C01354=45.159,-60.870,74.567,176.7508,4.4791,-13103.4286
C01355=49.709,-66.782,76.575,176.2813,5.1235,-13103.3379
C01356=53.692,-72.396,77.551,177.2844,5.6222,-13103.4378
C01357=54.731,-78.373,78.062,-179.5514,3.9310,-13105.0719
C01358=52.567,-83.926,78.476,-178.8613,1.5505,-13107.9391
C01359=47.632,-87.904,78.891,-179.8889,0.0607,-13111.5483
C01360=41.489,-90.984,79.163,-179.9865,0.0062,-13115.4869
C01361=34.998,-93.673,79.163,-179.9861,0.0052,-13119.5134
C01362=28.477,-95.839,78.891,-179.8785,0.0356,-13123.4515
C01363=22.174,-96.515,78.476,-178.0988,-0.2913,-13127.0610
C01364=16.717,-94.118,78.062,-176.9018,-2.4653,-13129.9283
C01365=13.226,-89.158,77.551,-177.9343,-5.8891,-13131.5621
C01366=12.073,-82.372,76.575,-179.0007,-6.2410,-13131.6617
C01367=11.109,-74.974,74.567,-179.1263,-5.4571,-13131.5717
C01368=10.239,-68.282,71.901,-179.2620,-4.2251,-13131.4719
C01369=9.406,-63.206,69.285,-179.7171,-1.2730,-13131.5356
C01370=7.959,-60.221,67.386,163.5021,14.7072,-13132.4712
C01371=4.772,-59.445,66.632,146.2352,3.2869,-13135.4104
C01372=2.097,-59.523,66.599,145.3553,-1.6722,-13137.9823
C01373=0.000,-59.554,66.621,145.3415,-0.0009,-13140.0000
C01374=0.000,-59.554,66.621,145.3415,-0.0009,-13140.0000
C01375=-2.096,-59.523,66.599,145.3552,1.6732,-13142.0167
C01376=-4.772,-59.445,66.632,146.2360,-3.2897,-13144.5896
C01377=-7.959,-60.222,67.386,163.5025,-14.7072,-13147.5286
C01378=-9.406,-63.206,69.285,-179.7171,1.2730,-13148.4644
C01379=-10.239,-68.282,71.901,-179.2620,4.2251,-13148.5281
C01380=-11.109,-74.974,74.567,-179.1263,5.4571,-13148.4283
C01381=-12.073,-82.372,76.575,-179.0007,6.2410,-13148.3383
C01382=-13.226,-89.158,77.551,-177.9343,5.8891,-13148.4379
C01383=-16.717,-94.118,78.062,-176.9018,2.4653,-13150.0717
C01384=-22.174,-96.515,78.476,-178.0988,0.2913,-13152.9390
C01385=-28.477,-95.839,78.891,-179.8785,-0.0356,-13156.5485
C01386=-34.998,-93.673,79.163,-179.9861,-0.0052,-13160.4866
C01387=-41.489,-90.984,79.163,-179.9865,-0.0062,-13164.5131
C01388=-47.632,-87.904,78.891,-179.8889,-0.0607,-13168.4517
C01389=-52.567,-83.926,78.476,-178.8613,-1.5505,-13172.0609
C01390=-54.731,-78.373,78.062,-179.5514,-3.9310,-13174.9281
C01391=-53.692,-72.396,77.551,177.2844,-5.6222,-13176.5622
C01392=-49.709,-66.782,76.575,176.2813,-5.1235,-13176.6621
C01393=-45.159,-60.870,74.567,176.7508,-4.4791,-13176.5714
C01394=-41.042,-55.523,71.901,177.5304,-3.5105,-13176.4714
C01395=-38.042,-51.344,69.285,179.2998,-1.1002,-13176.5356
C01396=-36.955,-48.211,67.386,178.6352,21.5554,-13177.4711
C01397=-38.660,-45.408,66.632,156.6295,27.1736,-13180.4108
C01398=-40.607,-43.572,66.599,153.0121,25.0783,-13182.9827
C01399=-42.111,-42.111,66.621,153.9470,26.0519,-13185.0000
C01400=-43.571,-40.607,66.599,154.9223,26.9884,-13187.0166
C01401=-45.409,-38.659,66.632,152.8255,23.3682,-13189.5906
C01402=-48.211,-36.955,67.386,158.4450,1.3645,-13192.5289
C01403=-51.344,-38.042,69.285,-178.8998,0.7002,-13193.4644
C01404=-55.523,-41.042,71.901,-176.4895,2.4696,-13193.5286
C01405=-60.870,-45.159,74.567,-175.5209,3.2492,-13193.4286
C01406=-66.782,-49.709,76.575,-174.8765,3.7187,-13193.3379
C01407=-72.396,-53.692,77.551,-174.3778,2.7156,-13193.4378
C01408=-78.373,-54.731,78.062,-176.0690,-0.4486,-13195.0719
C01409=-83.926,-52.567,78.476,-178.4495,-1.1387,-13197.9391
C01410=-87.904,-47.632,78.891,-179.9393,-0.1111,-13201.5483
C01411=-90.984,-41.489,79.163,-179.9938,-0.0135,-13205.4869
C01412=-93.673,-34.998,79.163,-179.9948,-0.0139,-13209.5134
C01413=-95.839,-28.477,78.891,-179.9644,-0.1215,-13213.4515
C01414=-96.515,-22.174,78.476,179.7087,-1.9012,-13217.0610
C01415=-94.118,-16.717,78.062,177.5347,-3.0982,-13219.9283
C01416=-89.158,-13.226,77.551,174.1109,-2.0657,-13221.5621
C01417=-82.372,-12.073,76.575,173.7590,-0.9993,-13221.6617
C01418=-74.974,-11.109,74.567,174.5429,-0.8737,-13221.5717
C01419=-68.282,-10.239,71.901,175.7749,-0.7380,-13221.4719
C01420=-63.206,-9.406,69.285,178.7270,-0.2829,-13221.5356
C01421=-60.221,-7.959,67.386,-165.2928,16.4979,-13222.4712
C01422=-59.445,-4.772,66.632,-176.7131,33.7648,-13225.4104
C01423=-59.523,-2.097,66.599,178.3278,34.6447,-13227.9823
C01424=-59.554,0.000,66.621,179.9991,34.6585,-13230.0000
C01425=-59.523,2.096,66.599,-178.3268,34.6448,-13232.0167
C01426=-59.445,4.772,66.632,176.7103,33.7640,-13234.5896
C01427=-60.222,7.959,67.386,165.2928,16.4975,-13237.5286
C01428=-63.206,9.406,69.285,-178.7270,-0.2829,-13238.4644
C01429=-68.282,10.239,71.901,-175.7749,-0.7380,-13238.5281
C01430=-74.974,11.109,74.567,-174.5429,-0.8737,-13238.4283
C01431=-82.372,12.073,76.575,-173.7590,-0.9993,-13238.3383
C01432=-89.158,13.226,77.551,-174.1109,-2.0657,-13238.4379
C01433=-94.118,16.717,78.062,-177.5347,-3.0982,-13240.0717
C01434=-96.515,22.174,78.476,-179.7087,-1.9012,-13242.9390
C01435=-95.839,28.477,78.891,179.9644,-0.1215,-13246.5485
C01436=-93.673,34.998,79.163,179.9948,-0.0139,-13250.4866
C01437=-90.984,41.489,79.163,179.9938,-0.0135,-13254.5131
C01438=-87.904,47.632,78.891,179.9393,-0.1111,-13258.4517
C01439=-83.926,52.567,78.476,178.4495,-1.1387,-13262.0609
C01440=-78.373,54.731,78.062,176.0690,-0.4486,-13264.9281
C01441=-72.396,53.692,77.551,174.3778,2.7156,-13266.5622
C01442=-66.782,49.709,76.575,174.8765,3.7187,-13266.6621
C01443=-60.870,45.159,74.567,175.5209,3.2492,-13266.5714
C01444=-55.523,41.042,71.901,176.4895,2.4696,-13266.4714
C01445=-51.344,38.042,69.285,178.8998,0.7002,-13266.5356
C01446=-48.211,36.955,67.386,-158.4446,1.3648,-13267.4711
C01447=-45.408,38.660,66.632,-152.8264,23.3705,-13270.4108
C01448=-43.572,40.607,66.599,-154.9217,26.9879,-13272.9827
C01449=-42.111,42.111,66.621,-153.9481,26.0530,-13275.0000
C01450=-40.607,43.571,66.599,-153.0116,25.0777,-13277.0166
C01451=-38.659,45.409,66.632,-156.6318,27.1745,-13279.5906
C01452=-36.955,48.211,67.386,-178.6355,21.5550,-13282.5289
C01453=-38.042,51.344,69.285,-179.2998,-1.1002,-13283.4644
C01454=-41.042,55.523,71.901,-177.5304,-3.5105,-13283.5286
C01455=-45.159,60.870,74.567,-176.7508,-4.4791,-13283.4286
C01456=-49.709,66.782,76.575,-176.2813,-5.1235,-13283.3379
C01457=-53.692,72.396,77.551,-177.2844,-5.6222,-13283.4378
C01458=-54.731,78.373,78.062,179.5514,-3.9310,-13285.0719
C01459=-52.567,83.926,78.476,178.8613,-1.5505,-13287.9391
C01460=-47.632,87.904,78.891,179.8889,-0.0607,-13291.5483
C01461=-41.489,90.984,79.163,179.9865,-0.0062,-13295.4869
C01462=-34.998,93.673,79.163,179.9861,-0.0052,-13299.5134
C01463=-28.477,95.839,78.891,179.8785,-0.0356,-13303.4515
C01464=-22.174,96.515,78.476,178.0988,0.2913,-13307.0610
C01465=-16.717,94.118,78.062,176.9018,2.4653,-13309.9283
C01466=-13.226,89.158,77.551,177.9343,5.8891,-13311.5621
C01467=-12.073,82.372,76.575,179.0007,6.2410,-13311.6617
C01468=-11.109,74.974,74.567,179.1263,5.4571,-13311.5717
C01469=-10.239,68.282,71.901,179.2620,4.2251,-13311.4719
C01470=-9.406,63.206,69.285,179.7171,1.2730,-13311.5356
C01471=-7.959,60.222,67.386,-163.5025,-14.7072,-13312.4714
C01472=-4.772,59.445,66.632,-146.2360,-3.2897,-13315.4104
C01473=-2.096,59.523,66.599,-145.3552,1.6732,-13317.9833
C01474=0.000,59.554,66.621,-145.3415,-0.0009,-13320.0000
C01475=0.000,58.319,68.442,-146.3550,-0.0009,-13320.0000
C01476=1.984,58.291,68.419,-146.3668,-1.5596,-13321.9494
C01477=4.582,58.225,68.453,-147.3209,3.5043,-13324.4996
C01478=7.730,59.058,69.238,-164.9099,14.0649,-13327.4570
C01479=9.135,62.185,71.215,179.6644,-1.6099,-13328.3570
C01480=9.949,67.473,73.927,179.3067,-4.1423,-13328.3879
C01481=10.820,74.409,76.674,179.2045,-5.1449,-13328.2735
C01482=11.787,82.032,78.729,179.1118,-5.7669,-13328.1767
C01483=12.929,88.996,79.725,178.1562,-5.4103,-13328.2659
C01484=16.445,94.085,80.245,177.1832,-2.2811,-13329.9145
C01485=21.964,96.553,80.665,178.2682,-0.2736,-13332.8156
C01486=28.347,95.882,81.086,179.8893,0.0324,-13336.4700
C01487=34.955,93.690,81.363,179.9874,0.0047,-13340.4601
C01488=41.532,90.965,81.363,179.9877,0.0056,-13344.5401
C01489=47.755,87.843,81.086,179.8988,0.0554,-13348.5303
C01490=52.743,83.804,80.665,178.9686,1.4181,-13352.1847
C01491=54.900,78.157,80.245,179.6205,3.6025,-13355.0854
C01492=53.787,72.072,79.725,-177.4688,5.1275,-13356.7338
C01493=49.670,66.340,78.729,-176.5407,4.7091,-13356.8229
C01494=44.964,60.266,76.674,-176.9177,4.2028,-13356.7263
C01495=40.676,54.746,73.927,-177.5576,3.4203,-13356.6122
C01496=37.512,50.430,71.215,-179.0987,1.3757,-13356.6435
C01497=36.294,47.226,69.238,-179.2260,-20.1942,-13357.5429
C01498=37.931,44.411,68.453,-157.6922,-26.4224,-13360.5003
C01499=39.816,42.621,68.419,-153.9116,-24.2820,-13363.0512
C01500=41.238,41.238,68.442,-154.7977,-25.2012,-13365.0000
C01501=42.621,39.816,68.419,-155.7185,-26.0890,-13366.9488
C01502=44.412,37.931,68.453,-153.5766,-22.3055,-13369.5003
C01503=47.226,36.294,69.238,-159.8063,-0.7736,-13372.4571
C01504=50.430,37.512,71.215,178.6243,-0.9013,-13373.3565
C01505=54.746,40.676,73.927,176.5797,-2.4424,-13373.3878
C01506=60.266,44.964,76.674,175.7972,-3.0823,-13373.2737
C01507=66.340,49.670,78.729,175.2909,-3.4593,-13373.1771
C01508=72.072,53.787,79.725,174.8725,-2.5312,-13373.2662
C01509=78.157,54.900,80.245,176.3975,0.3795,-13374.9146
C01510=83.804,52.743,80.665,178.5819,1.0314,-13377.8153
C01511=87.843,47.755,81.086,179.9446,0.1012,-13381.4697
C01512=90.965,41.532,81.363,179.9944,0.0123,-13385.4599
C01513=93.690,34.955,81.363,179.9953,0.0126,-13389.5399
C01514=95.882,28.347,81.086,179.9676,0.1107,-13393.5300
C01515=96.553,21.964,80.665,-179.7264,1.7318,-13397.1844
C01516=94.085,16.445,80.245,-177.7189,2.8168,-13400.0855
C01517=88.996,12.929,79.725,-174.5897,1.8438,-13401.7341
C01518=82.032,11.787,78.729,-174.2331,0.8882,-13401.8233
C01519=74.409,10.820,76.674,-174.8551,0.7955,-13401.7265
C01520=67.473,9.949,73.927,-175.8577,0.6933,-13401.6121
C01521=62.185,9.135,71.215,-178.3901,0.3356,-13401.6430
C01522=59.058,7.730,69.238,165.9351,-15.0901,-13402.5430
C01523=58.225,4.582,68.453,176.4957,-32.6791,-13405.5004
C01524=58.291,1.984,68.419,-178.4404,-33.6332,-13408.0506
C01525=58.319,0.000,68.442,-179.9991,-33.6450,-13410.0000
C01526=58.291,-1.983,68.419,178.4394,-33.6332,-13411.9484
C01527=58.225,-4.583,68.453,-176.4929,-32.6783,-13414.5006
C01528=59.058,-7.730,69.238,-165.9352,-15.0895,-13417.4570
C01529=62.185,-9.135,71.215,178.3901,0.3356,-13418.3570
C01530=67.473,-9.949,73.927,175.8577,0.6933,-13418.3879
C01531=74.409,-10.820,76.674,174.8551,0.7955,-13418.2735
C01532=82.032,-11.787,78.729,174.2331,0.8882,-13418.1767
C01533=88.996,-12.929,79.725,174.5897,1.8438,-13418.2659
C01534=94.085,-16.445,80.245,177.7189,2.8168,-13419.9145
C01535=96.553,-21.964,80.665,179.7264,1.7318,-13422.8156
C01536=95.882,-28.347,81.086,-179.9676,0.1107,-13426.4700
C01537=93.690,-34.955,81.363,-179.9953,0.0126,-13430.4601
C01538=90.965,-41.532,81.363,-179.9944,0.0123,-13434.5401
C01539=87.843,-47.755,81.086,-179.9446,0.1012,-13438.5303
C01540=83.804,-52.743,80.665,-178.5819,1.0314,-13442.1847
C01541=78.157,-54.900,80.245,-176.3975,0.3795,-13445.0854
C01542=72.072,-53.787,79.725,-174.8725,-2.5312,-13446.7338
C01543=66.340,-49.670,78.729,-175.2909,-3.4593,-13446.8229
C01544=60.266,-44.964,76.674,-175.7972,-3.0823,-13446.7263
C01545=54.746,-40.676,73.927,-176.5797,-2.4424,-13446.6122
C01546=50.430,-37.512,71.215,-178.6243,-0.9013,-13446.6435
C01547=47.226,-36.294,69.238,159.8058,-0.7740,-13447.5429
C01548=44.411,-37.931,68.453,153.5776,-22.3078,-13450.5003
C01549=42.621,-39.816,68.419,155.7180,-26.0884,-13453.0512
C01550=41.238,-41.238,68.442,154.7988,-25.2023,-13455.0000
C01551=39.816,-42.621,68.419,153.9110,-24.2815,-13456.9488
C01552=37.931,-44.412,68.453,157.6945,-26.4234,-13459.5003
C01553=36.294,-47.226,69.238,179.2264,-20.1937,-13462.4571
C01554=37.512,-50.430,71.215,179.0987,1.3757,-13463.3565
C01555=40.676,-54.746,73.927,177.5576,3.4203,-13463.3878
C01556=44.964,-60.266,76.674,176.9177,4.2028,-13463.2737
C01557=49.670,-66.340,78.729,176.5407,4.7091,-13463.1771
C01558=53.787,-72.072,79.725,177.4688,5.1275,-13463.2662
C01559=54.900,-78.157,80.245,-179.6205,3.6025,-13464.9146
C01560=52.743,-83.804,80.665,-178.9686,1.4181,-13467.8153
C01561=47.755,-87.843,81.086,-179.8988,0.0554,-13471.4697
C01562=41.532,-90.965,81.363,-179.9877,0.0056,-13475.4599
C01563=34.955,-93.690,81.363,-179.9874,0.0047,-13479.5399
C01564=28.347,-95.882,81.086,-179.8893,0.0324,-13483.5300
C01565=21.964,-96.553,80.665,-178.2682,-0.2736,-13487.1844
C01566=16.445,-94.085,80.245,-177.1832,-2.2811,-13490.0855
C01567=12.929,-88.996,79.725,-178.1562,-5.4103,-13491.7341
C01568=11.787,-82.032,78.729,-179.1118,-5.7669,-13491.8233
C01569=10.820,-74.409,76.674,-179.2045,-5.1449,-13491.7265
C01570=9.949,-67.473,73.927,-179.3067,-4.1423,-13491.6121
C01571=9.135,-62.185,71.215,-179.6644,-1.6099,-13491.6430
C01572=7.730,-59.058,69.238,164.9099,14.0649,-13492.5430
C01573=4.582,-58.225,68.453,147.3209,3.5043,-13495.5004
C01574=1.984,-58.291,68.419,146.3668,-1.5596,-13498.0506
C01575=0.000,-58.319,68.442,146.3550,-0.0009,-13500.0000
C01576=0.000,-58.319,68.442,146.3550,-0.0009,-13500.0000
C01577=-1.983,-58.291,68.419,146.3668,1.5606,-13501.9484
C01578=-4.583,-58.225,68.453,147.3217,-3.5071,-13504.5006
C01579=-7.730,-59.058,69.238,164.9105,-14.0648,-13507.4570
C01580=-9.135,-62.185,71.215,-179.6644,1.6099,-13508.3570
C01581=-9.949,-67.473,73.927,-179.3067,4.1423,-13508.3879
C01582=-10.820,-74.409,76.674,-179.2045,5.1449,-13508.2735
C01583=-11.787,-82.032,78.729,-179.1118,5.7669,-13508.1767
C01584=-12.929,-88.996,79.725,-178.1562,5.4103,-13508.2659
C01585=-16.445,-94.085,80.245,-177.1832,2.2811,-13509.9145
C01586=-21.964,-96.553,80.665,-178.2682,0.2736,-13512.8156
C01587=-28.347,-95.882,81.086,-179.8893,-0.0324,-13516.4700
C01588=-34.955,-93.690,81.363,-179.9874,-0.0047,-13520.4601
C01589=-41.532,-90.965,81.363,-179.9877,-0.0056,-13524.5401
C01590=-47.755,-87.843,81.086,-179.8988,-0.0554,-13528.5303
C01591=-52.743,-83.804,80.665,-178.9686,-1.4181,-13532.1847
C01592=-54.900,-78.157,80.245,-179.6205,-3.6025,-13535.0854
C01593=-53.787,-72.072,79.725,177.4688,-5.1275,-13536.7338
C01594=-49.670,-66.340,78.729,176.5407,-4.7091,-13536.8229
C01595=-44.964,-60.266,76.674,176.9177,-4.2028,-13536.7263
C01596=-40.676,-54.746,73.927,177.5576,-3.4203,-13536.6122
C01597=-37.512,-50.430,71.215,179.0987,-1.3757,-13536.6435
C01598=-36.294,-47.226,69.238,179.2260,20.1942,-13537.5429
C01599=-37.931,-44.411,68.453,157.6922,26.4224,-13540.5003
C01600=-39.816,-42.621,68.419,153.9116,24.2820,-13543.0512
C01601=-41.238,-41.238,68.442,154.7977,25.2012,-13545.0000
C01602=-42.621,-39.816,68.419,155.7185,26.0890,-13546.9488
C01603=-44.412,-37.931,68.453,153.5766,22.3055,-13549.5003
C01604=-47.226,-36.294,69.238,159.8063,0.7736,-13552.4571
C01605=-50.430,-37.512,71.215,-178.6243,0.9013,-13553.3565
C01606=-54.746,-40.676,73.927,-176.5797,2.4424,-13553.3878
C01607=-60.266,-44.964,76.674,-175.7972,3.0823,-13553.2737
C01608=-66.340,-49.670,78.729,-175.2909,3.4593,-13553.1771
C01609=-72.072,-53.787,79.725,-174.8725,2.5312,-13553.2662
C01610=-78.157,-54.900,80.245,-176.3975,-0.3795,-13554.9146
C01611=-83.804,-52.743,80.665,-178.5819,-1.0314,-13557.8153
C01612=-87.843,-47.755,81.086,-179.9446,-0.1012,-13561.4697
C01613=-90.965,-41.532,81.363,-179.9944,-0.0123,-13565.4599
C01614=-93.690,-34.955,81.363,-179.9953,-0.0126,-13569.5399
C01615=-95.882,-28.347,81.086,-179.9676,-0.1107,-13573.5300
C01616=-96.553,-21.964,80.665,179.7264,-1.7318,-13577.1844
C01617=-94.085,-16.445,80.245,177.7189,-2.8168,-13580.0855
C01618=-88.996,-12.929,79.725,174.5897,-1.8438,-13581.7341
C01619=-82.032,-11.787,78.729,174.2331,-0.8882,-13581.8233
C01620=-74.409,-10.820,76.674,174.8551,-0.7955,-13581.7265
C01621=-67.473,-9.949,73.927,175.8577,-0.6933,-13581.6121
C01622=-62.185,-9.135,71.215,178.3901,-0.3356,-13581.6430
C01623=-59.058,-7.730,69.238,-165.9351,15.0901,-13582.5430
C01624=-58.225,-4.582,68.453,-176.4957,32.6791,-13585.5004
C01625=-58.291,-1.984,68.419,178.4404,33.6332,-13588.0506
C01626=-58.319,0.000,68.442,179.9991,33.6450,-13590.0000
C01627=-58.291,1.983,68.419,-178.4394,33.6332,-13591.9484
C01628=-58.225,4.583,68.453,176.4929,32.6783,-13594.5006
C01629=-59.058,7.730,69.238,165.9352,15.0895,-13597.4570
C01630=-62.185,9.135,71.215,-178.3901,-0.3356,-13598.3570
C01631=-67.473,9.949,73.927,-175.8577,-0.6933,-13598.3879
C01632=-74.409,10.820,76.674,-174.8551,-0.7955,-13598.2735
C01633=-82.032,11.787,78.729,-174.2331,-0.8882,-13598.1767
C01634=-88.996,12.929,79.725,-174.5897,-1.8438,-13598.2659
C01635=-94.085,16.445,80.245,-177.7189,-2.8168,-13599.9145
C01636=-96.553,21.964,80.665,-179.7264,-1.7318,-13602.8156
C01637=-95.882,28.347,81.086,179.9676,-0.1107,-13606.4700
C01638=-93.690,34.955,81.363,179.9953,-0.0126,-13610.4601
C01639=-90.965,41.532,81.363,179.9944,-0.0123,-13614.5401
C01640=-87.843,47.755,81.086,179.9446,-0.1012,-13618.5303
C01641=-83.804,52.743,80.665,178.5819,-1.0314,-13622.1847
C01642=-78.157,54.900,80.245,176.3975,-0.3795,-13625.0854
C01643=-72.072,53.787,79.725,174.8725,2.5312,-13626.7338
C01644=-66.340,49.670,78.729,175.2909,3.4593,-13626.8229
C01645=-60.266,44.964,76.674,175.7972,3.0823,-13626.7263
C01646=-54.746,40.676,73.927,176.5797,2.4424,-13626.6122
C01647=-50.430,37.512,71.215,178.6243,0.9013,-13626.6435
C01648=-47.226,36.294,69.238,-159.8058,0.7740,-13627.5429
C01649=-44.411,37.931,68.453,-153.5776,22.3078,-13630.5003
C01650=-42.621,39.816,68.419,-155.7180,26.0884,-13633.0512
C01651=-41.238,41.238,68.442,-154.7988,25.2023,-13635.0000
C01652=-39.816,42.621,68.419,-153.9110,24.2815,-13636.9488
C01653=-37.931,44.412,68.453,-157.6945,26.4234,-13639.5003
C01654=-36.294,47.226,69.238,-179.2264,20.1937,-13642.4571
C01655=-37.512,50.430,71.215,-179.0987,-1.3757,-13643.3565
C01656=-40.676,54.746,73.927,-177.5576,-3.4203,-13643.3878
C01657=-44.964,60.266,76.674,-176.9177,-4.2028,-13643.2737
C01658=-49.670,66.340,78.729,-176.5407,-4.7091,-13643.1771
C01659=-53.787,72.072,79.725,-177.4688,-5.1275,-13643.2662
C01660=-54.900,78.157,80.245,179.6205,-3.6025,-13644.9146
C01661=-52.743,83.804,80.665,178.9686,-1.4181,-13647.8153
C01662=-47.755,87.843,81.086,179.8988,-0.0554,-13651.4697
C01663=-41.532,90.965,81.363,179.9877,-0.0056,-13655.4599
C01664=-34.955,93.690,81.363,179.9874,-0.0047,-13659.5399
C01665=-28.347,95.882,81.086,179.8893,-0.0324,-13663.5300
C01666=-21.964,96.553,80.665,178.2682,0.2736,-13667.1844
C01667=-16.445,94.085,80.245,177.1832,2.2811,-13670.0855
C01668=-12.929,88.996,79.725,178.1562,5.4103,-13671.7341
C01669=-11.787,82.032,78.729,179.1118,5.7669,-13671.8233
C01670=-10.820,74.409,76.674,179.2045,5.1449,-13671.7265
C01671=-9.949,67.473,73.927,179.3067,4.1423,-13671.6121
C01672=-9.135,62.185,71.215,179.6644,1.6099,-13671.6430
C01673=-7.730,59.058,69.238,-164.9105,-14.0648,-13672.5430
C01674=-4.583,58.225,68.453,-147.3217,-3.5071,-13675.4994
C01675=-1.983,58.291,68.419,-146.3668,1.5606,-13678.0516
C01676=0.000,58.319,68.442,-146.3550,-0.0009,-13680.0000
C01677=0.000,57.118,70.285,-147.5034,-0.0009,-13680.0000
C01678=1.874,57.094,70.261,-147.5130,-1.4410,-13681.8799
C01679=4.398,57.039,70.297,-148.5403,3.6784,-13684.4091
C01680=7.507,57.930,71.114,-166.2856,13.3384,-13687.3837
C01681=8.875,61.204,73.167,179.6344,-1.8648,-13688.2508
C01682=9.674,66.709,75.971,179.3569,-3.9987,-13688.2514
C01683=10.553,73.885,78.794,179.2847,-4.7758,-13688.1286
C01684=11.527,81.722,80.892,179.2219,-5.2319,-13688.0287
C01685=12.662,88.851,81.904,178.3832,-4.8674,-13688.1105
C01686=16.202,94.056,82.431,177.4937,-2.0609,-13689.7738
C01687=21.776,96.587,82.857,178.4589,-0.2498,-13692.7052
C01688=28.231,95.920,83.283,179.9016,0.0287,-13696.4001
C01689=34.916,93.705,83.562,179.9888,0.0041,-13700.4362
C01690=41.570,90.949,83.562,179.9892,0.0050,-13704.5637
C01691=47.863,87.788,83.283,179.9101,0.0492,-13708.5997
C01692=52.900,83.695,82.857,179.0867,1.2664,-13712.2952
C01693=55.051,77.964,82.431,179.6845,3.2279,-13715.2262
C01694=53.873,71.781,81.904,-177.6947,4.5839,-13716.8889
C01695=49.635,65.937,80.892,-176.8436,4.2522,-13716.9711
C01696=44.783,59.707,78.794,-177.1234,3.8847,-13716.8716
C01697=40.330,54.011,75.971,-177.6240,3.2832,-13716.7487
C01698=37.003,49.553,73.167,-178.9395,1.5772,-13716.7500
C01699=35.654,46.271,71.114,-179.7188,-18.7891,-13717.6160
C01700=37.223,43.442,70.297,-158.8350,-25.5520,-13720.5914
C01701=39.047,41.697,70.261,-154.9186,-23.3867,-13723.1202
C01702=40.388,40.388,70.285,-155.7518,-24.2471,-13725.0000
C01703=41.696,39.047,70.261,-156.6139,-25.0820,-13726.8791
C01704=43.443,37.223,70.297,-154.4471,-21.1627,-13729.4092
C01705=46.271,35.654,71.114,-161.2114,-0.2808,-13732.3840
C01706=49.553,37.003,73.167,178.4228,-1.0605,-13733.2500
C01707=54.011,40.330,75.971,176.7168,-2.3760,-13733.2513
C01708=59.707,44.783,78.794,176.1153,-2.8766,-13733.1284
C01709=65.937,49.635,80.892,175.7478,-3.1564,-13733.0289
C01710=71.781,53.873,81.904,175.4161,-2.3053,-13733.1111
C01711=77.964,55.051,82.431,176.7721,0.3155,-13734.7738
C01712=83.695,52.900,82.857,178.7336,0.9133,-13737.7048
C01713=87.788,47.863,83.283,179.9508,0.0899,-13741.4003
C01714=90.949,41.570,83.562,179.9950,0.0108,-13745.4363
C01715=93.705,34.916,83.562,179.9959,0.0112,-13749.5638
C01716=95.920,28.231,83.283,179.9713,0.0984,-13753.5999
